(* Logix 5000 project; controller PRU vendor 1 type 14 code 107 rev 20.13; software revision 20.01; part 3 of 17 *)
(* tags used below, declared in another part *)
   LEFT_AUTO_PCNT_SETPOINT : REAL;
   Revision : DINT;
   VFD_3_Current : DINT;

ADD_ON_INSTRUCTION Totalize   (* revision 1.0, ExecuteEnableInFalse *)
// This instruction takes a flow signal (mL/min) and converts it to a total volume (mL)
VAR_INPUT
   FlowMeterCV : REAL; {required}
END_VAR
VAR_IN_OUT
   TotalVolume : REAL; {required}
END_VAR
VAR_INPUT
   FlowValve : BOOL; {required}
END_VAR
VAR_OUTPUT
   VolAddedLast : REAL; {access Read Only, visible}
END_VAR
VAR
   TOT_02 : TOTALIZER := (In := 2.289028, TimeBase := 1, Gain := 1.0, ProgProgReq := 1, ProgStopReq := 1, ProgResetReq := 1, OversampleDT := 0.5, RTSTime := 1, OldTotal := 413.70062, ProgOper := 1, ProgResetDone := 1, TargetFlag := 1, TargetDev1Flag := 1, TargetDev2Flag := 1, DeltaT := 0.001);
   BNOT_01 : FBD_BOOLEAN_NOT := (In := 1);
   __l01CE45141B44CC5A : REAL;
   __l01CE49331B44B276 : BOOL;
END_VAR

ROUTINE EnableInFalse   (* ladder *)
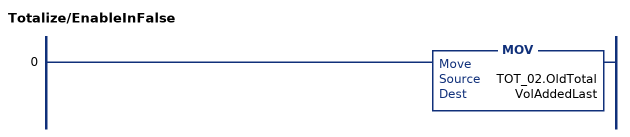
   0: MOV(TOT_02.OldTotal,VolAddedLast);
END_ROUTINE

ROUTINE Logic   (* function block diagram *)
   SHEET 1
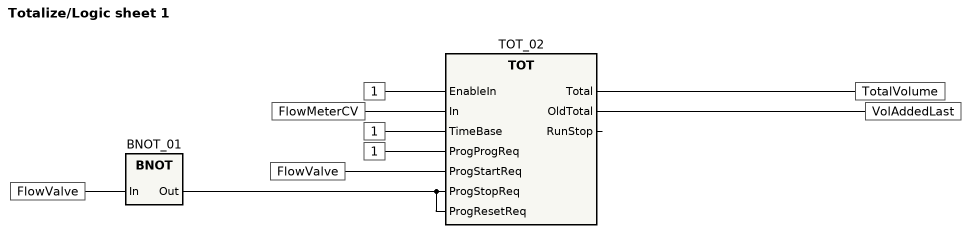
   BNOT_01 : BNOT(In := FlowValve);
   TOT_02 : TOT(EnableIn := 1, In := FlowMeterCV, TimeBase := 1, ProgProgReq := 1, ProgStartReq := FlowValve, ProgStopReq := BNOT_01.Out, ProgResetReq := BNOT_01.Out);   // unwired pins: RunStop
   TotalVolume := TOT_02.Total;
   VolAddedLast := TOT_02.OldTotal;
END_ROUTINE
END_ADD_ON_INSTRUCTION

ADD_ON_INSTRUCTION VFD_Motor_Control   (* revision 1.2, vendor Deterministic Systems, Inc. *)
// VFD Motor Control
VAR_INPUT
   IN_HARD_STOP : BOOL; {required}
   IN_HMI_STOP_PB : BOOL; {required}
   IN_RUN_INTERLOCK_1 : BOOL; {required}
   IN_RUN_INTERLOCK_2 : BOOL; {required}
   IN_RUN_INTERLOCK_3 : BOOL; {required}
   IN_VFD_IS_READY : BOOL; {required}
   IN_HMI_OFF_PB : BOOL; {required}   // Pushbutton.
   IN_HMI_MAINT_PB : BOOL; {required}   // Pushbutton.
   IN_HMI_SEMI_PB : BOOL; {required}   // Pushbutton.
   IN_HMI_AUTO_PB : BOOL; {required}   // Pushbutton.
   IN_HMI_JOG_FWD_PB : BOOL; {required}   // Pushbutton.
   IN_HMI_JOG_REV_PB : BOOL; {required}   // Pushbutton.
   IN_HMI_FWD_PB : BOOL; {required}   // Pushbutton.
   IN_HMI_REV_PB : BOOL; {required}   // Pushbutton.
   IN_HMI_AUTO_START_PB : BOOL; {required}
   IN_CURRENT_PROCESS_SEQUENCER_STEP : INT; {required}
   IN_PROCESS_SEQUENCER_AUTO_START_STEP : INT; {required}
   IN_PROCESS_SEQUENCER_AUTO_STOP_STEP : INT; {required}
   IN_HMI_SEMI_SPEED_SETPOINT_PCNT : REAL; {required}
   IN_AUTO_SPEED_SETPOINT_PERCENT : REAL; {required}
   IN_VFD_SPEED_SCALE : REAL := 6.0; {required}
   IN_VFD_ACTUAL_FREQ : REAL; {required}   // Direct from VFD.
   IN_VFD_IS_RUNNING : BOOL; {required}
END_VAR
VAR_OUTPUT
   OUT_HARD_STOPPED : BOOL; {access Read Only, required}
   OUT_OFF_MODE_ION : BOOL; {access Read Only, required}
   OUT_MAINT_MODE_ION : BOOL; {access Read Only, required}
   OUT_SEMI_MODE_ION : BOOL; {access Read Only, required}
   OUT_AUTO_MODE_ION : BOOL; {access Read Only, required}
   OUT_MODE : INT; {access Read Only, required}
   OUT_VFD_STOP_COMMAND : BOOL; {access Read Only, required}   // Direct to VFD.
   OUT_FWD_COMMAND : BOOL; {access Read Only, required}   // Direct to VFD.
   OUT_REV_COMMAND : BOOL; {access Read Only, required}   // Direct to VFD.
   OUT_JOG_COMMAND : BOOL; {access Read Only, required}   // Direct to VFD.
   OUT_VFD_RUN_COMMAND : BOOL; {access Read Only, required}   // Direct to VFD.
   OUT_CMD_RUN_ENABLED : BOOL; {access Read Only, required}   // Auto or Semi
   OUT_START_CMD_AUTO : BOOL; {access None, required}
   OUT_VFD_SPEED_SETPOINT_COMMAND : DINT; {access Read Only, required}   // Direct to VFD.
   OUT_VFD_ACTUAL_SPEED_PERCENT : REAL; {access Read Only, required}
   OUT_RUNNING_BON : BOOL; {access Read Only, required}
   OUT_RUNNING_BOF : BOOL; {access Read Only, required}
END_VAR
VAR
   AUTO_PB_ONS : BOOL; {access None}
   SEMI_PB_ONS : BOOL; {access None}
   MAINT_PB_ONS : BOOL; {access None}
   JOG_FWD_TON : TIMER := (PRE := 30000); {access None}
   LOCAL_AUTO_SETPOINT_PERCENT : REAL; {access None}
   RUNNING_TON : TIMER := (PRE := 1000); {access None}
   RUNNING_TOF : TIMER := (PRE := 1000); {access None}
END_VAR

ROUTINE Logic   (* ladder *)
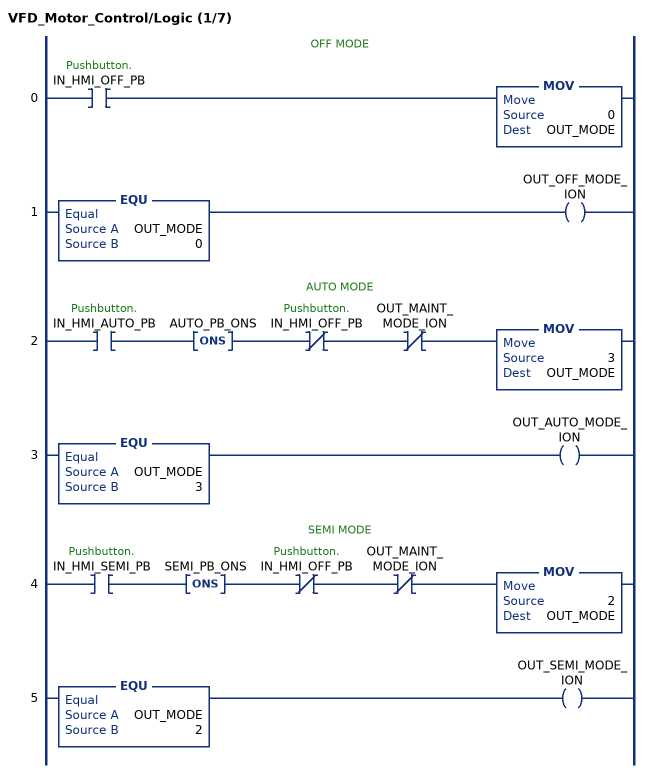
   // OFF MODE
   0: XIC(IN_HMI_OFF_PB)MOV(0,OUT_MODE);
   1: EQU(OUT_MODE,0)OTE(OUT_OFF_MODE_ION);
   // AUTO MODE
   2: XIC(IN_HMI_AUTO_PB)ONS(AUTO_PB_ONS)XIO(IN_HMI_OFF_PB)XIO(OUT_MAINT_MODE_ION)MOV(3,OUT_MODE);
   3: EQU(OUT_MODE,3)OTE(OUT_AUTO_MODE_ION);
   // SEMI MODE
   4: XIC(IN_HMI_SEMI_PB)ONS(SEMI_PB_ONS)XIO(IN_HMI_OFF_PB)XIO(OUT_MAINT_MODE_ION)MOV(2,OUT_MODE);
   5: EQU(OUT_MODE,2)OTE(OUT_SEMI_MODE_ION);
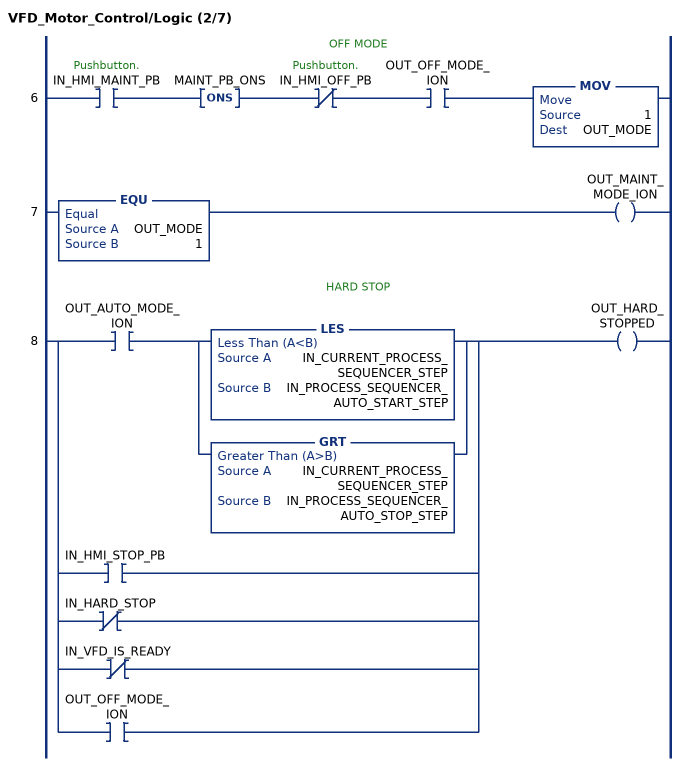
   // OFF MODE
   6: XIC(IN_HMI_MAINT_PB)ONS(MAINT_PB_ONS)XIO(IN_HMI_OFF_PB)XIC(OUT_OFF_MODE_ION)MOV(1,OUT_MODE);
   7: EQU(OUT_MODE,1)OTE(OUT_MAINT_MODE_ION);
   // HARD STOP
   8: [XIC(OUT_AUTO_MODE_ION) [LES(IN_CURRENT_PROCESS_SEQUENCER_STEP,IN_PROCESS_SEQUENCER_AUTO_START_STEP) ,GRT(IN_CURRENT_PROCESS_SEQUENCER_STEP,IN_PROCESS_SEQUENCER_AUTO_STOP_STEP) ] ,XIC(IN_HMI_STOP_PB) ,XIO(IN_HARD_STOP) ,XIO(IN_VFD_IS_READY) ,XIC(OUT_OFF_MODE_ION) ]OTE(OUT_HARD_STOPPED);
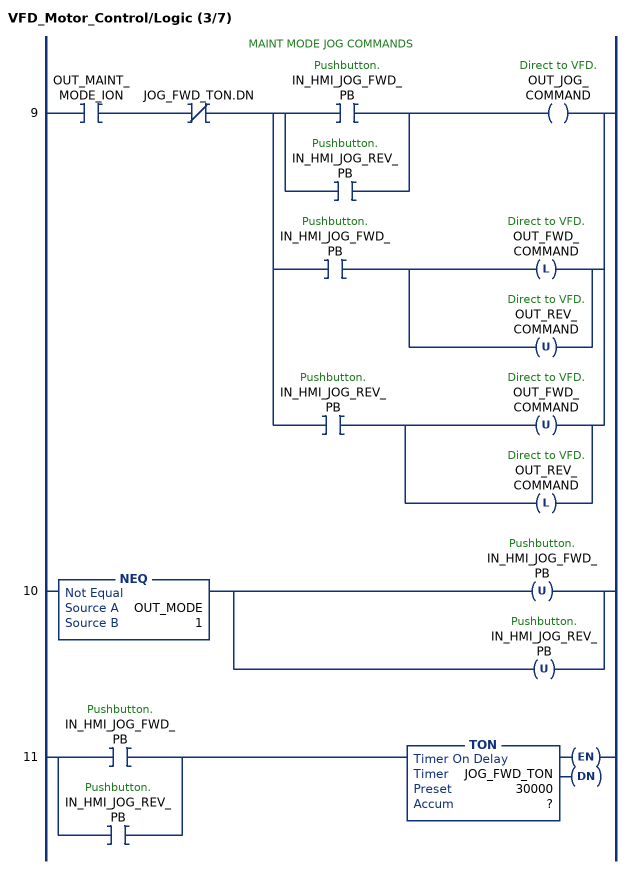
   // MAINT MODE JOG COMMANDS
   9: XIC(OUT_MAINT_MODE_ION)XIO(JOG_FWD_TON.DN)[[XIC(IN_HMI_JOG_FWD_PB) ,XIC(IN_HMI_JOG_REV_PB) ] OTE(OUT_JOG_COMMAND) ,XIC(IN_HMI_JOG_FWD_PB) [OTL(OUT_FWD_COMMAND) ,OTU(OUT_REV_COMMAND) ] ,XIC(IN_HMI_JOG_REV_PB) [OTU(OUT_FWD_COMMAND) ,OTL(OUT_REV_COMMAND) ] ];
   10: NEQ(OUT_MODE,1)[OTU(IN_HMI_JOG_FWD_PB) ,OTU(IN_HMI_JOG_REV_PB) ];
   11: [XIC(IN_HMI_JOG_FWD_PB) ,XIC(IN_HMI_JOG_REV_PB) ]TON(JOG_FWD_TON,?,?);
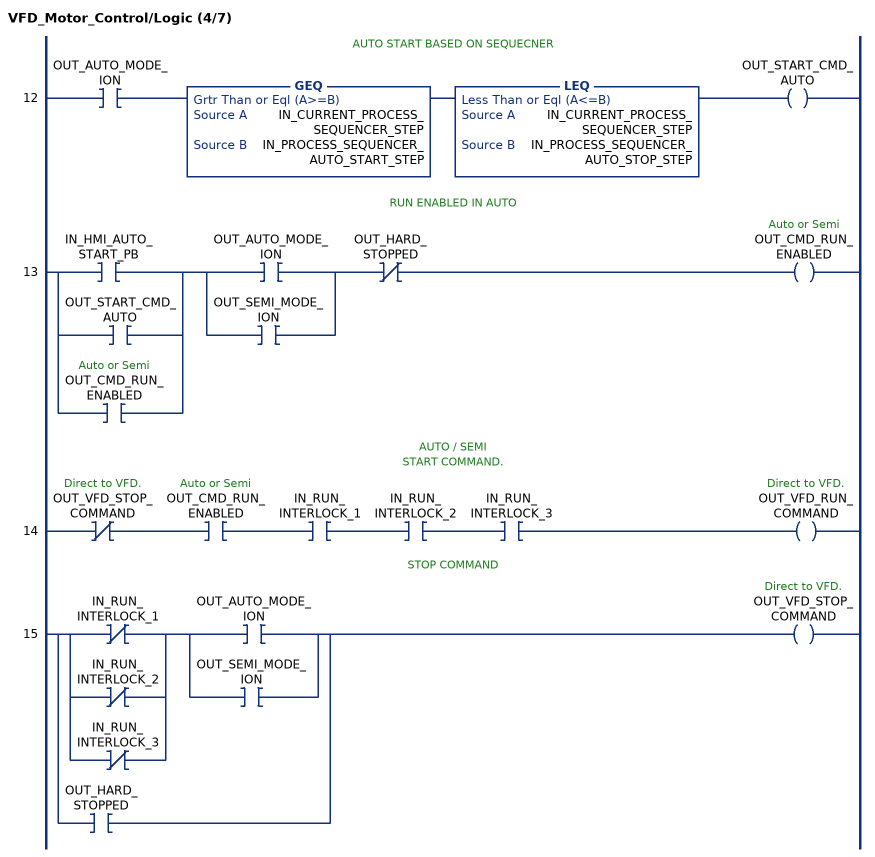
   // AUTO START BASED ON SEQUECNER
   12: XIC(OUT_AUTO_MODE_ION)GEQ(IN_CURRENT_PROCESS_SEQUENCER_STEP,IN_PROCESS_SEQUENCER_AUTO_START_STEP)LEQ(IN_CURRENT_PROCESS_SEQUENCER_STEP,IN_PROCESS_SEQUENCER_AUTO_STOP_STEP)OTE(OUT_START_CMD_AUTO);
   // RUN ENABLED IN AUTO
   13: [[XIC(IN_HMI_AUTO_START_PB) ,XIC(OUT_START_CMD_AUTO) ] ,XIC(OUT_CMD_RUN_ENABLED) ][XIC(OUT_AUTO_MODE_ION) ,XIC(OUT_SEMI_MODE_ION) ]XIO(OUT_HARD_STOPPED)OTE(OUT_CMD_RUN_ENABLED);
   // AUTO / SEMI
   // START COMMAND.
   14: XIO(OUT_VFD_STOP_COMMAND)XIC(OUT_CMD_RUN_ENABLED)XIC(IN_RUN_INTERLOCK_1)XIC(IN_RUN_INTERLOCK_2)XIC(IN_RUN_INTERLOCK_3)OTE(OUT_VFD_RUN_COMMAND);
   // STOP COMMAND
   15: [[XIO(IN_RUN_INTERLOCK_1) ,XIO(IN_RUN_INTERLOCK_2) ,XIO(IN_RUN_INTERLOCK_3) ] [XIC(OUT_AUTO_MODE_ION) ,XIC(OUT_SEMI_MODE_ION) ] ,XIC(OUT_HARD_STOPPED) ]OTE(OUT_VFD_STOP_COMMAND);
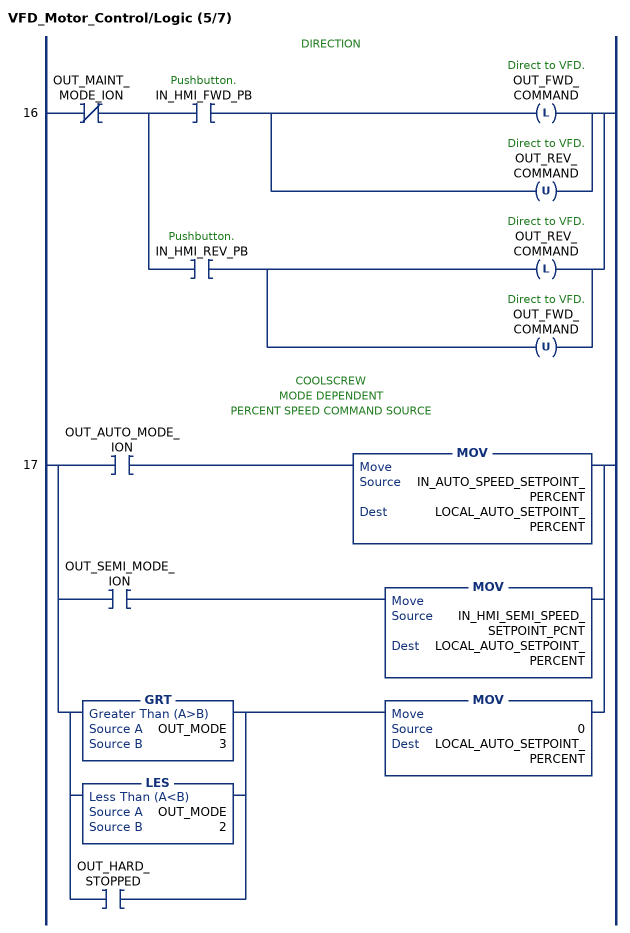
   // DIRECTION
   16: XIO(OUT_MAINT_MODE_ION)[XIC(IN_HMI_FWD_PB) [OTL(OUT_FWD_COMMAND) ,OTU(OUT_REV_COMMAND) ] ,XIC(IN_HMI_REV_PB) [OTL(OUT_REV_COMMAND) ,OTU(OUT_FWD_COMMAND) ] ];
   // COOLSCREW
   // MODE DEPENDENT
   // PERCENT SPEED COMMAND SOURCE
   17: [XIC(OUT_AUTO_MODE_ION) MOV(IN_AUTO_SPEED_SETPOINT_PERCENT,LOCAL_AUTO_SETPOINT_PERCENT) ,XIC(OUT_SEMI_MODE_ION) MOV(IN_HMI_SEMI_SPEED_SETPOINT_PCNT,LOCAL_AUTO_SETPOINT_PERCENT) ,[GRT(OUT_MODE,3) ,LES(OUT_MODE,2) ,XIC(OUT_HARD_STOPPED) ] MOV(0,LOCAL_AUTO_SETPOINT_PERCENT) ];
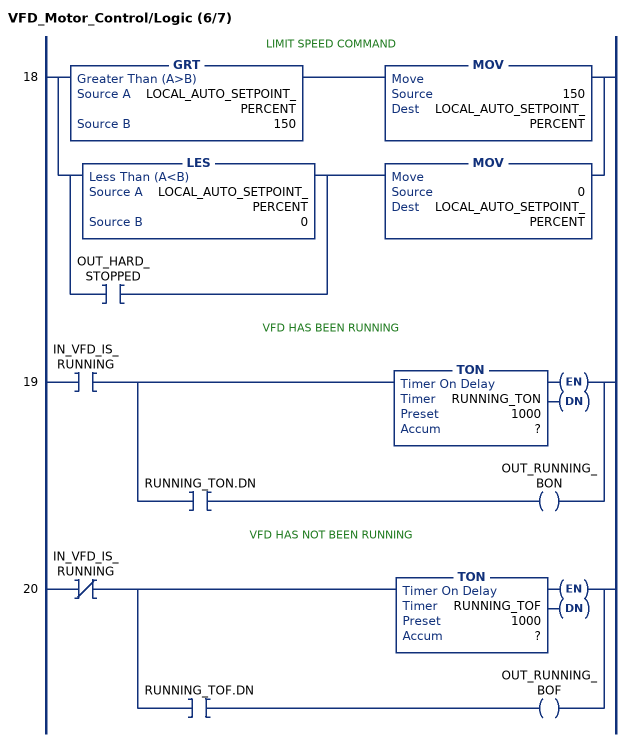
   // LIMIT SPEED COMMAND
   18: [GRT(LOCAL_AUTO_SETPOINT_PERCENT,150) MOV(150,LOCAL_AUTO_SETPOINT_PERCENT) ,[LES(LOCAL_AUTO_SETPOINT_PERCENT,0) ,XIC(OUT_HARD_STOPPED) ] MOV(0,LOCAL_AUTO_SETPOINT_PERCENT) ];
   // VFD HAS BEEN RUNNING
   19: XIC(IN_VFD_IS_RUNNING)[TON(RUNNING_TON,?,?) ,XIC(RUNNING_TON.DN) OTE(OUT_RUNNING_BON) ];
   // VFD HAS NOT BEEN RUNNING
   20: XIO(IN_VFD_IS_RUNNING)[TON(RUNNING_TOF,?,?) ,XIC(RUNNING_TOF.DN) OTE(OUT_RUNNING_BOF) ];
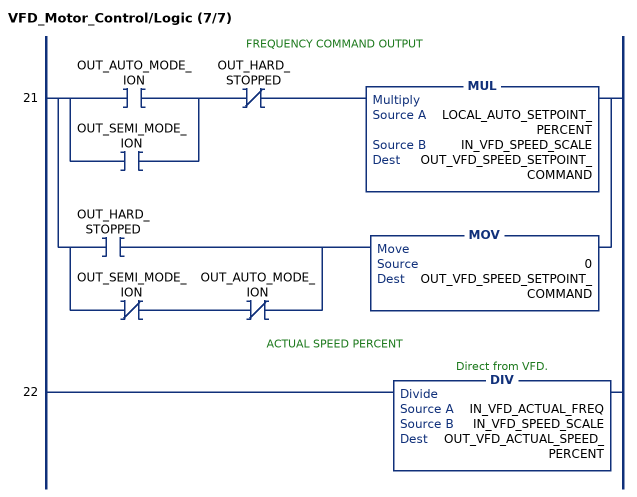
   // FREQUENCY COMMAND OUTPUT
   21: [[XIC(OUT_AUTO_MODE_ION) ,XIC(OUT_SEMI_MODE_ION) ] XIO(OUT_HARD_STOPPED) MUL(LOCAL_AUTO_SETPOINT_PERCENT,IN_VFD_SPEED_SCALE,OUT_VFD_SPEED_SETPOINT_COMMAND) ,[XIC(OUT_HARD_STOPPED) ,XIO(OUT_SEMI_MODE_ION) XIO(OUT_AUTO_MODE_ION) ] MOV(0,OUT_VFD_SPEED_SETPOINT_COMMAND) ];
   // ACTUAL SPEED PERCENT
   22: DIV(IN_VFD_ACTUAL_FREQ,IN_VFD_SPEED_SCALE,OUT_VFD_ACTUAL_SPEED_PERCENT);
END_ROUTINE
END_ADD_ON_INSTRUCTION

VAR_GLOBAL   (* controller tags *)
   ABS_ENCODER_ERROR_MINUS : REAL := 58.63318;
   ABS_ENCODER_ERROR_PLUS : REAL := 72.63318;
   ACCEL_DECEL_RAMP : REAL := 200.0;   // VFD Accel/Decel ramp rate * 10ms ie 100 * 10ms = 1sec
   ACTUAL_FWD_ION : BOOL := 1;
   ACTUAL_ILLEGAL_ION : BOOL;
   ACTUAL_REV_ION : BOOL;
   AFI : BOOL;
   Agilyx_KnifeGateIgnorePB : BOOL := 1;
   AI0_CALCULATED : REAL := 0.06;
   AI0_WF : DSi_WF50 := (IN_VALUE := 6.0, OUT_VALUE := 6.0);
   AI10_CALCULATED : REAL := 0.08;
   AI10_WF : DSi_WF50 := (IN_VALUE := 8.0, OUT_VALUE := 7.5);
   AI11_CALCULATED : REAL := 0.03;
   AI11_WF : DSi_WF50 := (OUT_VALUE := 2.88);
   AI12_CALCULATED : REAL := 0.089999996;
   AI12_WF : DSi_WF50 := (IN_VALUE := 12.0, OUT_VALUE := 9.12);
   AI13_CALCULATED : REAL := 18.56;
   AI13_WF : DSi_WF50 := (IN_VALUE := 1693.0, OUT_VALUE := 1813.78);
   AI14_CALCULATED : REAL := 19.279999;
   AI14_WF : DSi_WF50 := (IN_VALUE := 2256.0, OUT_VALUE := 2126.92);
   AI15_CALCULATED : REAL := -5.0;
   AI15_WF : DSi_WF50 := (IN_VALUE := -500.0, OUT_VALUE := -500.0);
   AI16_CALCULATED : REAL := 3.2;
   AI16_WF : DSi_WF50 := (IN_VALUE := -500.0, OUT_VALUE := -500.0);
   AI1_CALCULATED : REAL := 0.099999994;
   AI1_WF : DSi_WF50 := (IN_VALUE := 10.0, OUT_VALUE := 10.0);
   AI2_CALCULATED : REAL := 0.11;
   AI2_WF : DSi_WF50 := (IN_VALUE := 11.0, OUT_VALUE := 11.34);
   AI3_CALCULATED : REAL := 0.06;
   AI3_WF : DSi_WF50 := (IN_VALUE := 6.0, OUT_VALUE := 6.16);
   AI4_CALCULATED : REAL := 0.06;
   AI4_WF : DSi_WF50 := (IN_VALUE := 6.0, OUT_VALUE := 6.0);
   AI5_CALCULATED : REAL := 0.01;
   AI5_WF : DSi_WF50 := (IN_VALUE := 4.0, OUT_VALUE := 2.12);
   AI6_CALCULATED : REAL := 2.44;
   AI6_WF : DSi_WF50 := (IN_VALUE := 82.0, OUT_VALUE := 344.3);
   AI7_CALCULATED : REAL := 2.31;
   AI7_WF : DSi_WF50 := (IN_VALUE := 672.0, OUT_VALUE := 235.98);
   AI8_CALCULATED : REAL := 2.04;
   AI8_WF : DSi_WF50 := (IN_VALUE := 111.0, OUT_VALUE := 309.82);
   AI9_CALCULATED : REAL := 0.02;
   AI9_WF : DSi_WF50 := (IN_VALUE := -1.0, OUT_VALUE := 1.74);
   AI_0 : AI_1769_IF4 := (IN_ANALOG_INPUT_RAW := 6, IN_Ai_Hi_Scale := 100.0, IN_HMI_Ai_FORCE_VALUE := 3.0, OUT_Ai_Calc := 0.06, OUT_ANALOG_OUTPUT := 0.06);
   AI_0_FILTERED : DINT := 6;
   AI_1 : AI_1769_IF4 := (IN_ANALOG_INPUT_RAW := 10, IN_Ai_Hi_Scale := 100.0, IN_HMI_Ai_FORCE_VALUE := 3.0, OUT_Ai_Calc := 0.099999994, OUT_ANALOG_OUTPUT := 0.099999994);
   AI_10 : AI_1769_IF4 := (IN_ANALOG_INPUT_RAW := 8, IN_Ai_Hi_Scale := 100.0, OUT_Ai_Calc := 0.08, OUT_ANALOG_OUTPUT := 0.08);
   AI_10_FILTERED : REAL := 8.4;
   AI_11 : AI_1769_IF4 := (IN_ANALOG_INPUT_RAW := 2, IN_Ai_Hi_Scale := 100.0, IN_HMI_Ai_FORCE_VALUE := 33.0, OUT_Ai_Calc := 0.02, OUT_ANALOG_OUTPUT := 0.02);
   AI_11_FILTERED : REAL := 0.86;
   AI_12 : AI_1769_IF4 := (IN_ANALOG_INPUT_RAW := 9, IN_Ai_Hi_Scale := 100.0, IN_HMI_Ai_FORCE_VALUE := 42.0, OUT_Ai_Calc := 0.089999996, OUT_ANALOG_OUTPUT := 0.089999996);
   AI_12_FILTERED : REAL := 8.58;
   AI_13 : AI_1769_IF4 := (IN_ANALOG_INPUT_RAW := 1847, IN_Ai_Hi_Scale := 100.0, IN_HMI_Ai_FORCE_VALUE := 35.0, OUT_Ai_Calc := 18.47, OUT_ANALOG_OUTPUT := 18.47);
   AI_13_FILTERED : REAL := 1851.82;
   AI_14 : AI_1769_IF4 := (IN_ANALOG_INPUT_RAW := 1925, IN_Ai_Hi_Scale := 100.0, IN_HMI_Ai_FORCE_VALUE := 42.0, OUT_Ai_Calc := 19.25, OUT_ANALOG_OUTPUT := 19.25);
   AI_14_FILTERED : REAL := 1941.48;
   AI_15 : AI_1769_IF4 := (IN_ANALOG_INPUT_RAW := -500, IN_Ai_Hi_Scale := 100.0, IN_HMI_Ai_FORCE_VALUE := 37.0, OUT_Ai_Calc := -5.0, OUT_ANALOG_OUTPUT := -5.0);
   AI_15_FILTERED : REAL := -500.0;
   AI_16 : AI_1769_IF4 := (IN_ANALOG_INPUT_RAW := -500, IN_Ai_Lo_Scale := 4.0, IN_Ai_Hi_Scale := 20.0, IN_HMI_Ai_FORCE_VALUE := 50.0, OUT_Ai_Calc := 3.2, OUT_ANALOG_OUTPUT := 3.2);
   AI_16_DATA : REAL := 3.2;
   AI_16_FILTERED : REAL := -500.0;
   AI_1_FILTERED : REAL := 10.0;
   AI_2 : AI_1769_IF4 := (IN_ANALOG_INPUT_RAW := 11, IN_Ai_Hi_Scale := 100.0, IN_HMI_Ai_FORCE_VALUE := 3.0, OUT_Ai_Calc := 0.11, OUT_ANALOG_OUTPUT := 0.11);
   AI_2_FILTERED : REAL := 11.1;
   AI_3 : AI_1769_IF4 := (IN_ANALOG_INPUT_RAW := 7, IN_Ai_Hi_Scale := 100.0, IN_HMI_Ai_FORCE_VALUE := 3.0, OUT_Ai_Calc := 0.07, OUT_ANALOG_OUTPUT := 0.07);
   AI_3_FILTERED : REAL := 6.32;
   AI_4 : AI_1769_IF4 := (IN_ANALOG_INPUT_RAW := 6, IN_Ai_Hi_Scale := 100.0, IN_HMI_Ai_FORCE_VALUE := 3.0, OUT_Ai_Calc := 0.06, OUT_ANALOG_OUTPUT := 0.06);
   AI_4_FILTERED : REAL := 6.26;
   AI_5 : AI_1769_IF4 := (IN_ANALOG_INPUT_RAW := 2, IN_Ai_Hi_Scale := 100.0, IN_HMI_Ai_FORCE_VALUE := 3.0, OUT_Ai_Calc := 0.02, OUT_ANALOG_OUTPUT := 0.02);
   AI_5_FILTERED : REAL := 1.48;
   AI_6 : AI_1769_IF4 := (IN_ANALOG_INPUT_RAW := 333, IN_Ai_Hi_Scale := 100.0, IN_HMI_Ai_FORCE_VALUE := 3.0, OUT_Ai_Calc := 3.33, OUT_ANALOG_OUTPUT := 3.33);
   AI_6_FILTERED : REAL := 236.58;
   AI_7 : AI_1769_IF4 := (IN_ANALOG_INPUT_RAW := 224, IN_Ai_Hi_Scale := 100.0, IN_HMI_Ai_FORCE_VALUE := 3.0, OUT_Ai_Calc := 2.24, OUT_ANALOG_OUTPUT := 2.24);
   AI_7_FILTERED : REAL := 233.06;
   AI_8 : AI_1769_IF4 := (IN_ANALOG_INPUT_RAW := 275, IN_Ai_Hi_Scale := 100.0, IN_HMI_Ai_FORCE_VALUE := 10.0, OUT_Ai_Calc := 2.75, OUT_ANALOG_OUTPUT := 2.75);
   AI_8_FILTERED : REAL := 198.48;
   AI_9 : AI_1769_IF4 := (IN_ANALOG_INPUT_RAW := 2, IN_Ai_Hi_Scale := 100.0, IN_HMI_Ai_FORCE_VALUE := 15.0, OUT_Ai_Calc := 0.02, OUT_ANALOG_OUTPUT := 0.02);
   AI_9_FILTERED : REAL := 1.4;
   AlarmMaster : DINT;
        .0   // MESSAGE ALARM bit.0
        .1   // WARNING ALARM bit.1
        .2   // CSS_START_DISABLE bit.2
        .3   // PRU_START_DISABLE bit.3
        .4   // PRU_RUN_DISABLE bit.4
   AlarmMasterDisable : BOOL;
   AlarmMasterResetTON : TIMER := (PRE := 1000, ACC := 689, EN := 1, TT := 1);
   AlarmResetPB : BOOL;
   ALL_AUTO_IOK : BOOL := 1;   // All equipment is in Auto Mode.
   ALL_DRIVES_ARE_CMD_FWD : BOOL := 1;
   ALL_DRIVES_ARE_READY : BOOL := 1;
   ALL_SHUTDOWN_FAULTS_IOK : BOOL := 1;
   AUTO_DISCHARGE_CYCLE_ION : BOOL := 1;   // Proces Sequencer (4-13)
   AUTO_FWD_CMD : BOOL;
   AUTO_FWD_CMD_GON : BOOL := 1;
   AUTO_FWD_CMD_GON_VALUE : DINT := 3;
   AUTO_FWD_CMD_VALUE : DINT;
   AUTO_SHUTDOWN_ENABLE : BOOL := 1;
   CALC_SPARE_AO_CMD : REAL := 50.0;
   CENTERING_BON : BOOL;
   CENTERING_BON_ONS : BOOL;
   CENTERING_BON_SS : BOOL;
   CENTERING_ERROR : REAL;
   CENTERING_ERROR_NOW : REAL;
   CENTERING_ERROR_WAS : REAL;
   CENTERING_ONS : BOOL;
   CENTERING_SS : BOOL;
   CENTERING_TON : TIMER := (PRE := 1000);
   CHANGING_TOTE : BOOL;
   CHANGING_TOTE_1 : BOOL;
   CHANGING_TOTE_2 : BOOL;
   CHANGING_TOTE_3 : BOOL;
   CHANGING_TOTE_4 : BOOL;
   CHANGING_TOTE_5 : BOOL;
   CLEARING_PYROLIZER_TIME_REMAINING_SEC : REAL := 60.0;
   CLEARING_PYROLIZER_TIME_REMAINING_TEMP : REAL := 60000.0;
   CLEARING_PYROLIZER_TIMER : TIMER := (PRE := 60000);
   CMD_LEFT_SCREW_START : BOOL;
   CMD_LEFT_SCREW_STOP : BOOL;
   CMD_RIGHT_SCREW_START : BOOL;
   CMD_RIGHT_SCREW_STOP : BOOL;
   CONTROLLED_STOP : BOOL;
   COOL_FOR_MOTOR_STOP : BOOL;
   COOL_MESSAGE_FON1 : TIMER := (PRE := 1000);
   COOL_MESSAGE_FON2 : TIMER := (PRE := 1000, ACC := 248, EN := 1, TT := 1);
   COOL_VFD_Message : MESSAGE;
        MessageParameters(ServiceCode := 16#000e, DestinationTag := VFD_3_Current, ...)
   COOLSCREW : VFD := (MODE := 3, SPEED_SETPOINT_SEMI := 40.0, SPEED_SETPOINT_AUTO := 40.0, INTERLOCK_1 := 1, INTERLOCK_2 := 1, INTERLOCK_3 := 1, ACTUAL_SPEED := 40.0, ACTUAL_SPEED_CONVERSION_FACTOR := 6.0, MODE_AUTO_ION := 1, VFD_BEEN_ON := 1, CMD_AUTO_RUN_ENABLED := 1, CMD_AUTO_STARTED := 1);
   CR0_CON1_HTR1_GON : BOOL := 1;   // ZONE 1 (L1,L2,L3)
   CR0_CON1_HTR1_LON : BOOL := 1;   // AUTO LOGIC - ZONE 1 HEATER CONTACTOR
   CR1_CON2_HTR2_GON : BOOL := 1;   // ZONE 2 (L1,L2,L3)
   CR1_CON2_HTR2_LON : BOOL := 1;   // AUTO LOGIC - ZONE 2 HEATER CONTACTOR
   CR2_CON3_HTR3_GON : BOOL := 1;   // ZONE 3 (L1,L2,L3)
   CR2_CON3_HTR3_LON : BOOL := 1;   // AUTO LOGIC - ZONE 3 HEATER CONTACTOR
   CR3_CON4_HTR4_GON : BOOL := 1;   // ZONE 4 (L1) ZONE 5 (L2) ZONE 6 (L3)
   CR3_CON4_HTR4_LON : BOOL := 1;   // AUTO LOGIC - ZONES 4-6 HEATER CONTACTOR
   CR4_CON5_HTR5_GON : BOOL := 1;   // ZONE 7 (L1) ZONE 8 (L2) ZONE 9 (L3)
   CR4_CON5_HTR5_LON : BOOL := 1;   // AUTO LOGIC - ZONES 7-9 HEATER CONTACTOR
   CR5_CON1_SAFETY_GON : BOOL := 1;
   CR5_CON1_SAFETY_LON : BOOL := 1;
   CR6_CON2_SAFETY_GON : BOOL := 1;
   CR6_CON2_SAFETY_LON : BOOL := 1;
   CR7_VFD_DRYERL_GON : BOOL := 1;
   CR7_VFD_DRYERL_LON : BOOL := 1;
   CR8_VFD_DRYERR_GON : BOOL;
   CR8_VFD_DRYERR_LON : BOOL;
   CSS_CommsLoss_TMR : TIMER := (PRE := 60000, EN := 1, TT := 1);
   CSS_CommsLossAlm : BOOL;
   CSS_CommsWarning_TMR : TIMER := (PRE := 5000);
   CSS_CommsWarningAlm : BOOL;
   CSS_PLC_Seconds_Temp : DINT := 6;
   CSS_Status_Data : PLCStatusData := (PLCSenonds := 12, AlarmMaster := 2, Status[0] := 403, Status[1] := 723, Status[2] := 623, Status[3] := -1872, Status[4] := -1995, Status[5] := -2109, Status[6] := 8414, Status[7] := -4146, Status[8] := -4000);
   CYCLE_ION_DELAY1_TON : TIMER := (PRE := 2000, ACC := 2001, EN := 1, DN := 1);
   CYCLE_ION_DELAY2_TON : TIMER := (PRE := 2000, ACC := 2006, EN := 1, DN := 1);
   CYCLE_ION_DELAY3_TON : TIMER := (PRE := 2000, ACC := 2000, EN := 1, DN := 1);
   CYCLE_ION_DELAY4_TON : TIMER := (PRE := 2000, ACC := 2003, EN := 1, DN := 1);
   CYCLE_START_ONS : BOOL;
   CYCLE_START_SS : BOOL;   // Begin temperature ramp and hold heat cycle.
   DailyTotalResetPB : BOOL := 1;
   DATA_RECORD_INDEX : INT;
   DCS_ESTOP_ION : BOOL := 1;
   DI0_ION : BOOL := 1;
   DI10_ION : BOOL;
   DI11_ION : BOOL := 1;
   DI12_ION : BOOL;
   DI13_ION : BOOL := 1;
   DI14_ION : BOOL;
   DI15_ION : BOOL := 1;
   DI16_ION : BOOL;
   DI17_ION : BOOL;
   DI18_ION : BOOL := 1;
   DI19_ION : BOOL := 1;
   DI1_ION : BOOL := 1;
   DI20_ION : BOOL := 1;
   DI21_ION : BOOL;
   DI22_ION : BOOL := 1;
   DI23_ION : BOOL;
   DI24_ION : BOOL;
   DI25_ION : BOOL;
   DI26_ION : BOOL;
   DI27_ION : BOOL := 1;
   DI28_ION : BOOL;
   DI29_ION : BOOL;
   DI2_ION : BOOL := 1;
   DI30_ION : BOOL;
   DI31_ION : BOOL;
   DI3_ION : BOOL := 1;
   DI4_ION : BOOL := 1;
   DI5_ION : BOOL := 1;
   DI6_ION : BOOL := 1;
   DI7_ION : BOOL;
   DI8_ION : BOOL;
   DI9_ION : BOOL;
   DisableAllHeaters : BOOL;
   DRYER : DUAL_SCREW := (HMI_AUTO_SCREW_CMD_PCNT := 34.0, AUTO_SCREW_RIGHT_CMD_PCNT := 33.2266, LEFT_ENCODER_G := 3567, RIGHT_ENCODER_G := 559, LEFT_ENCODER_DEG_IS := 209.0039, RIGHT_ENCODER_DEG_IS := 274.7461, LEFT_AUTO_PCNT_SETPOINT := 34.0);
   DRYER_AUTO_MODE_PB_ONS : BOOL;
   DRYER_CENTER_STARTUP_MODE : BOOL;
   DRYER_CENTER_TON : TIMER := (PRE := 2000);
   DRYER_FWD_MODE : BOOL := 1;
   DRYER_IS_CENTERING : BOOL;
   DRYER_MAN_MODE_PB_ONS : BOOL;
   DRYER_MODE_AUTO : BOOL := 1;
   DRYER_MODE_OFF : BOOL;
   DRYER_ONS : BOOL := 1;
   DRYER_SEMIAUTO_MODE_PB_ONS : BOOL;
   DRYER_SHUTDOWN_FAULT_ION : BOOL;
   DRYERL_ACTUAL_SPEED : REAL := 16.0037;
   DRYERR_ACTUAL_SPEED : REAL := 12.937757;
   DUMMY_REAL : REAL;
   ENCODER_ACC : REAL := 14.501953;
   ENCODER_ERROR : REAL := 65.63008;
   ENCODER_OFFSET : REAL := -0.2;
   ENCODER_RATE : REAL := 14.501953;
   ESR_CONTACT_1_ION : BOOL := 1;
   ESR_CONTACT_2_ION : BOOL := 1;
   ESR_CONTACT_3_ION : BOOL;
   ESR_RESET_PB_ION : BOOL;
   ESTOP_PB_IOF : BOOL;   // E-STOP PUSHBUTTON IS PUSHED.
   FAULT : DINT[100];
        [9].0   // Changing Char Tote 1 Longer than 30 min
   FAULT_31_14_ONS : BOOL;
   FAULT_DRYERL_MSG_TON : TIMER := (PRE := 1000, ACC := 20, EN := 1, TT := 1);
   FAULT_DRYERR_MSG_TON : TIMER := (PRE := 1000, ACC := 20, EN := 1, TT := 1);
   FAULT_TIMER : TIMER[10000] := ([108].PRE := 5000, [109].PRE := 5000, [110].PRE := 5000, [111].PRE := 5000, [112].PRE := 5000, [113].PRE := 5000, [114].PRE := 5000, [115].PRE := 5000, [116].PRE := 5000, [117].PRE := 5000, [118].PRE := 5000, [119].PRE := 5000, [404].PRE := 5000, [500].PRE := 3000, [501].PRE := 3000, [600].PRE := 2000, [601].PRE := 2000, [602].PRE := 2000, [603].PRE := 2000, [604].PRE := 2000, [605].PRE := 2000, [606].PRE := 2000, [607].PRE := 2000, [608].PRE := 2000, [609].PRE := 2000, [610].PRE := 2000, [611].PRE := 2000, [612].PRE := 2000, [613].PRE := 2000, [614].PRE := 2000, [615].PRE := 2000, [616].PRE := 2000, [617].PRE := 2000, [618].PRE := 2000, [619].PRE := 2000, [620].PRE := 2000, [621].PRE := 2000, [622].PRE := 2000, [623].PRE := 2000, [624].PRE := 2000, [625].PRE := 2000, [626].PRE := 2000, [627].PRE := 2000, [628].PRE := 2000, [629].PRE := 2000, [630].PRE := 2000, [631].PRE := 2000, [700].PRE := 2000, [701].PRE := 2000, [702].PRE := 2000, [703].PRE := 2000, [704].PRE := 2000, [705].PRE := 2000, [706].PRE := 2000, [707].PRE := 2000, [708].PRE := 2000, [709].PRE := 2000, [710].PRE := 2000, [711].PRE := 2000, [712].PRE := 2000,
        [713].PRE := 2000, [714].PRE := 2000, [715].PRE := 2000, [716].PRE := 2000, [717].PRE := 2000, [718].PRE := 2000, [719].PRE := 2000, [720].PRE := 2000, [721].PRE := 2000, [722].PRE := 2000, [723].PRE := 2000, [724].PRE := 2000, [725].PRE := 2000, [726].PRE := 2000, [727].PRE := 2000, [728].PRE := 2000, [729].PRE := 2000, [730].PRE := 2000, [731].PRE := 2000, [800].PRE := 10000, [801].PRE := 10000, [3001].PRE := 1000, [3001].ACC := 10, [3001].EN := 1, [3001].TT := 1, [3002].PRE := 1000, [3004].PRE := 1500, [3006].PRE := 1500, [3007].PRE := 1500, [3010].PRE := 12000, [3011].PRE := 20, [3012].PRE := 20, [3014].PRE := 3000, [3016].PRE := 1000, [3017].PRE := 3000, [3019].PRE := 1500, [3020].PRE := 12000, [3021].PRE := 1500, [3022].PRE := 3000, [3025].PRE := 12000, [3026].PRE := 20, [3027].PRE := 20, [3029].PRE := 20, [3030].PRE := 2000, [3031].PRE := 1000, [3102].PRE := 1000, [3103].PRE := 1000, [3108].PRE := 5000, [3109].PRE := 5000, [3112].PRE := 100, [3113].PRE := 100, [3114].PRE := 1000, [4000].PRE := 2000, [4001].PRE := 2000, [4002].PRE := 2000, [4003].PRE := 2000, [4004].PRE := 2000, [4005].PRE := 2000, [4006].PRE := 2000, [4007].PRE := 2000,
        [4008].PRE := 2000, [4009].PRE := 2000, [4010].PRE := 2000, [4011].PRE := 2000, [4012].PRE := 2000, [4013].PRE := 2000, [4014].PRE := 2000, [4015].PRE := 2000, [4016].PRE := 2000, [4017].PRE := 2000, [4018].PRE := 2000, [4019].PRE := 2000, [4020].PRE := 2000, [4021].PRE := 2000, [4022].PRE := 2000, [4023].PRE := 2000, [4024].PRE := 2000, [4025].PRE := 2000, [4026].PRE := 2000, [4027].PRE := 2000, [4028].PRE := 2000, [4029].PRE := 2000, [4030].PRE := 2000, [4031].PRE := 2000, [5004].PRE := 2000, [5005].PRE := 20000, [5006].PRE := 3000, [5007].PRE := 3000, [5008].PRE := 2000, [5009].PRE := 10000, [5010].ACC := 4, [5010].EN := 1, [5010].DN := 1, [5800].PRE := 3000, [5801].PRE := 3000, [5802].PRE := 3000, [5803].PRE := 3000, [5804].PRE := 3000, [5805].PRE := 2000, [5806].PRE := 2000, [5807].PRE := 2000, [5808].PRE := 2000, [5809].PRE := 2000, [5810].PRE := 2000, [5811].PRE := 2000, [5812].PRE := 2000, [5813].PRE := 2000, [5814].PRE := 2000, [5815].PRE := 2000, [5816].PRE := 2000, [5817].PRE := 2000, [5818].PRE := 2000, [5819].PRE := 2000, [6500].PRE := 2000, [6501].PRE := 30000, [6502].PRE := 30000, [6503].PRE := 2000, [6600].PRE := 2000, [6601].PRE := 30000, [6602].PRE := 30000,
        [6603].PRE := 2000);
   FAULT_TIMER_3112_TmrExtended : BOOL;
   FAULT_TIMER_3112_TmrNormal : BOOL := 1;
   FAULTS_FA1_IOK : BOOL := 1;   // SYSTEM LEVEL FAULTS ARE OK.
   FAULTS_FA1A_IOK : BOOL := 1;   // MODULE FAULTS ARE OK.
   FAULTS_FA1B_IOK : BOOL := 1;   // STOP PUSHBUTTON FAULTS ARE OK.
   FAULTS_FA3_IOK : BOOL := 1;
   FAULTS_FA3A_IOK : BOOL := 1;   // SCREWS DRIVES NOT FAULTED.
   FAULTS_FA3B_IOK : BOOL := 1;   // ENCODERS NOT FAULTED.
   FAULTS_FA4_IOK : BOOL := 1;   // HI TEMP FAULTS ARE OK.
   FAULTS_FA4A_IOK : BOOL := 1;   // HIGH TEMPERATURE FAULTS ARE OK.
   FAULTS_FA5_IOK : BOOL := 1;
   FAULTS_FA5A_IOK : BOOL := 1;   // COOLING SCREW FAULTS ARE OK.
   FAULTS_FA5C_IOK : BOOL := 1;   // KG021 FAULTS ARE OK.
   FAULTS_FA5D_IOK : BOOL := 1;   // KG021 FAULTS ARE OK.
   FAULTS_FA6_IOK : BOOL := 1;   // HEATER FAULTS ARE OK.
   FAULTS_FA6A_IOK : BOOL := 1;
   FAULTS_FA6B_IOK : BOOL := 1;
   FEED_DWELL_DEG : INT;
   FEED_IS_DWELLING : BOOL := 1;
   FEED_SHOT_ENABLE_Enabled : BOOL := 1;
   FEED_SHOT_ENABLE_GON : BOOL;
   FEED_SHOT_ENABLE_GON_ONS : BOOL := 1;
   FEED_SHOT_ENABLE_GON_Tmr : TIMER := (PRE := 9999999, ACC := 12989);
   FEED_SHOT_ENABLE_GON_TmrONS : BOOL;
   FEED_SHOT_ENABLE_GON_TmrONS1 : BOOL;
   FEED_SHOT_ENABLE_GON_TmrONS2 : BOOL := 1;
   FEED_SHOT_ENABLE_ONS : BOOL := 1;
   FEED_SHOT_ENABLE_ONSN : BOOL;
   FEED_SHOT_ENABLE_SS : BOOL;
   FEED_SHOT_ENABLE_SSN : BOOL;
   FEED_TIME : REAL := 45.0;
   FEED_TIME_OFF : TIMER := (PRE := 45000);
   FEED_TIME_OFF_DSEC : REAL := 4000.0;
   FEED_TIME_OFF_REM : REAL := 45.0;
   FEED_TIME_OFF_REM_TEMP : REAL := 45000.0;
   FEED_TIME_OFF_SEC : REAL := 45.0;
   FEED_TIME_ON : TIMER;
   FEED_TIME_ON_REM : REAL;
   FEED_TIME_ON_REM_TEMP : REAL;
   FEED_TIME_ON_SEC : REAL;
   FEED_TRIGGER : BOOL := 1;
   FEED_UNWIND_THRESHOLD : INT := 145;
   FINISH_PROCESS_TIME_REMAINING_SEC : REAL := 120.0;
   FINISH_PROCESS_TIME_REMAINING_TEMP : REAL := 120000.0;
   FINISH_PROCESS_TIMER : TIMER := (PRE := 120000);
   FIRST_CYCLE : BOOL;
   FS0101_ION : BOOL := 1;   // LOW FLOW SWITCH - INLET AND DISCHARGE PURGE
   FS0102H_ION : BOOL := 1;   // HIGH FLOW SWITCH - DISCHARGE END SHAFT SEAL
   FS0102L_ION : BOOL := 1;   // LOW FLOW SWITCH - DISCHARGE END SHAFT SEAL
   FS0103H_ION : BOOL := 1;   // HIGH FLOW SWITCH - CHAMBER END INLET SEALS
   FS0103L_ION : BOOL := 1;   // LOW FLOW SWITCH - CHAMBER END INLET SEALS
   FS0201_ION : BOOL;   // LOW FLOW SWITCH - KG021 PURGE
   FS0202_ION : BOOL := 1;   // LOW FLOW SWITCH - KG022 PURGE
   FS0203H_ION : BOOL := 1;   // HIGH FLOW SWITCH - COOLING SHAFT SEALS
   FS0203L_ION : BOOL := 1;   // LOW FLOW SWITCH - COOLING SHAFT SEALS
   FS0204_ION : BOOL := 1;   // LOW FLOW SWITCH - COOLING SCREW COOLING WATER
   FWD_CMD_BON : TIMER := (PRE := 1500, ACC := 1506, EN := 1, DN := 1);
   FWD_SCAN_COUNT : DINT := 12989;
   FWD_SCAN_COUNTING : DINT := 2532;
   FWD_SCAN_SEC : REAL := 12.989;
   GRAY : REAL[4097] := ([1] := 0.087890625, [2] := 0.26367188, [3] := 0.17578125, [4] := 0.6152344, [5] := 0.52734375, [6] := 0.3515625, [7] := 0.43945312, [8] := 1.3183594, [9] := 1.2304688, [10] := 1.0546875, [11] := 1.1425781, [12] := 0.703125, [13] := 0.7910156, [14] := 0.9667969, [15] := 0.87890625, [16] := 2.7246094, [17] := 2.6367188, [18] := 2.4609375, [19] := 2.5488281, [20] := 2.109375, [21] := 2.1972656, [22] := 2.3730469, [23] := 2.2851562, [24] := 1.40625, [25] := 1.4941406, [26] := 1.6699219, [27] := 1.5820312, [28] := 2.0214844, [29] := 1.9335938, [30] := 1.7578125, [31] := 1.8457031, [32] := 5.5371094, [33] := 5.4492188, [34] := 5.2734375, [35] := 5.361328, [36] := 4.921875, [37] := 5.0097656, [38] := 5.185547, [39] := 5.0976562, [40] := 4.21875, [41] := 4.3066406, [42] := 4.482422, [43] := 4.3945312, [44] := 4.8339844, [45] := 4.7460938, [46] := 4.5703125, [47] := 4.658203, [48] := 2.8125, [49] := 2.9003906, [50] := 3.0761719, [51] := 2.9882812, [52] := 3.4277344, [53] := 3.3398438, [54] := 3.1640625, [55] := 3.2519531, [56] := 4.1308594, [57] := 4.0429688, [58] := 3.8671875, [59] := 3.9550781, [60] := 3.515625,
        [61] := 3.6035156, [62] := 3.7792969, [63] := 3.6914062, [64] := 11.162109, [65] := 11.074219, [66] := 10.8984375, [67] := 10.986328, [68] := 10.546875, [69] := 10.634766, [70] := 10.810547, [71] := 10.722656, [72] := 9.84375, [73] := 9.931641, [74] := 10.107422, [75] := 10.019531, [76] := 10.458984, [77] := 10.371094, [78] := 10.1953125, [79] := 10.283203, [80] := 8.4375, [81] := 8.525391, [82] := 8.701172, [83] := 8.613281, [84] := 9.052734, [85] := 8.964844, [86] := 8.7890625, [87] := 8.876953, [88] := 9.755859, [89] := 9.667969, [90] := 9.4921875, [91] := 9.580078, [92] := 9.140625, [93] := 9.228516, [94] := 9.404297, [95] := 9.316406, [96] := 5.625, [97] := 5.7128906, [98] := 5.888672, [99] := 5.8007812, [100] := 6.2402344, [101] := 6.1523438, [102] := 5.9765625, [103] := 6.064453, [104] := 6.9433594, [105] := 6.8554688, [106] := 6.6796875, [107] := 6.767578, [108] := 6.328125, [109] := 6.4160156, [110] := 6.591797, [111] := 6.5039062, [112] := 8.349609, [113] := 8.261719, [114] := 8.0859375, [115] := 8.173828, [116] := 7.734375, [117] := 7.8222656, [118] := 7.998047, [119] := 7.9101562, [120] := 7.03125,
        [121] := 7.1191406, [122] := 7.294922, [123] := 7.2070312, [124] := 7.6464844, [125] := 7.5585938, [126] := 7.3828125, [127] := 7.470703, [128] := 22.41211, [129] := 22.324219, [130] := 22.148438, [131] := 22.236328, [132] := 21.796875, [133] := 21.884766, [134] := 22.060547, [135] := 21.972656, [136] := 21.09375, [137] := 21.18164, [138] := 21.357422, [139] := 21.269531, [140] := 21.708984, [141] := 21.621094, [142] := 21.445312, [143] := 21.533203, [144] := 19.6875, [145] := 19.77539, [146] := 19.951172, [147] := 19.863281, [148] := 20.302734, [149] := 20.214844, [150] := 20.039062, [151] := 20.126953, [152] := 21.00586, [153] := 20.917969, [154] := 20.742188, [155] := 20.830078, [156] := 20.390625, [157] := 20.478516, [158] := 20.654297, [159] := 20.566406, [160] := 16.875, [161] := 16.96289, [162] := 17.138672, [163] := 17.050781, [164] := 17.490234, [165] := 17.402344, [166] := 17.226562, [167] := 17.314453, [168] := 18.19336, [169] := 18.105469, [170] := 17.929688, [171] := 18.017578, [172] := 17.578125, [173] := 17.666016, [174] := 17.841797, [175] := 17.753906, [176] := 19.59961, [177] := 19.511719, [178] := 19.335938, [179] := 19.423828, [180] := 18.984375,
        [181] := 19.072266, [182] := 19.248047, [183] := 19.160156, [184] := 18.28125, [185] := 18.36914, [186] := 18.544922, [187] := 18.457031, [188] := 18.896484, [189] := 18.808594, [190] := 18.632812, [191] := 18.720703, [192] := 11.25, [193] := 11.337891, [194] := 11.513672, [195] := 11.425781, [196] := 11.865234, [197] := 11.777344, [198] := 11.6015625, [199] := 11.689453, [200] := 12.568359, [201] := 12.480469, [202] := 12.3046875, [203] := 12.392578, [204] := 11.953125, [205] := 12.041016, [206] := 12.216797, [207] := 12.128906, [208] := 13.974609, [209] := 13.886719, [210] := 13.7109375, [211] := 13.798828, [212] := 13.359375, [213] := 13.447266, [214] := 13.623047, [215] := 13.535156, [216] := 12.65625, [217] := 12.744141, [218] := 12.919922, [219] := 12.832031, [220] := 13.271484, [221] := 13.183594, [222] := 13.0078125, [223] := 13.095703, [224] := 16.78711, [225] := 16.699219, [226] := 16.523438, [227] := 16.611328, [228] := 16.171875, [229] := 16.259766, [230] := 16.435547, [231] := 16.347656, [232] := 15.46875, [233] := 15.556641, [234] := 15.732422, [235] := 15.644531, [236] := 16.083984, [237] := 15.996094, [238] := 15.8203125, [239] := 15.908203, [240] := 14.0625,
        [241] := 14.150391, [242] := 14.326172, [243] := 14.238281, [244] := 14.677734, [245] := 14.589844, [246] := 14.4140625, [247] := 14.501953, [248] := 15.380859, [249] := 15.292969, [250] := 15.1171875, [251] := 15.205078, [252] := 14.765625, [253] := 14.853516, [254] := 15.029297, [255] := 14.941406, [256] := 44.91211, [257] := 44.82422, [258] := 44.648438, [259] := 44.73633, [260] := 44.296875, [261] := 44.384766, [262] := 44.560547, [263] := 44.472656, [264] := 43.59375, [265] := 43.68164, [266] := 43.85742, [267] := 43.76953, [268] := 44.208984, [269] := 44.121094, [270] := 43.945312, [271] := 44.033203, [272] := 42.1875, [273] := 42.27539, [274] := 42.45117, [275] := 42.36328, [276] := 42.802734, [277] := 42.714844, [278] := 42.539062, [279] := 42.626953, [280] := 43.50586, [281] := 43.41797, [282] := 43.242188, [283] := 43.33008, [284] := 42.890625, [285] := 42.978516, [286] := 43.154297, [287] := 43.066406, [288] := 39.375, [289] := 39.46289, [290] := 39.63867, [291] := 39.55078, [292] := 39.990234, [293] := 39.902344, [294] := 39.726562, [295] := 39.814453, [296] := 40.69336, [297] := 40.60547, [298] := 40.429688, [299] := 40.51758, [300] := 40.078125,
        [301] := 40.166016, [302] := 40.341797, [303] := 40.253906, [304] := 42.09961, [305] := 42.01172, [306] := 41.835938, [307] := 41.92383, [308] := 41.484375, [309] := 41.572266, [310] := 41.748047, [311] := 41.660156, [312] := 40.78125, [313] := 40.86914, [314] := 41.04492, [315] := 40.95703, [316] := 41.396484, [317] := 41.308594, [318] := 41.132812, [319] := 41.220703, [320] := 33.75, [321] := 33.83789, [322] := 34.01367, [323] := 33.92578, [324] := 34.365234, [325] := 34.277344, [326] := 34.101562, [327] := 34.189453, [328] := 35.06836, [329] := 34.98047, [330] := 34.804688, [331] := 34.89258, [332] := 34.453125, [333] := 34.541016, [334] := 34.716797, [335] := 34.628906, [336] := 36.47461, [337] := 36.38672, [338] := 36.210938, [339] := 36.29883, [340] := 35.859375, [341] := 35.947266, [342] := 36.123047, [343] := 36.035156, [344] := 35.15625, [345] := 35.24414, [346] := 35.41992, [347] := 35.33203, [348] := 35.771484, [349] := 35.683594, [350] := 35.507812, [351] := 35.595703, [352] := 39.28711, [353] := 39.19922, [354] := 39.023438, [355] := 39.11133, [356] := 38.671875, [357] := 38.759766, [358] := 38.935547, [359] := 38.847656, [360] := 37.96875,
        [361] := 38.05664, [362] := 38.23242, [363] := 38.14453, [364] := 38.583984, [365] := 38.496094, [366] := 38.320312, [367] := 38.408203, [368] := 36.5625, [369] := 36.65039, [370] := 36.82617, [371] := 36.73828, [372] := 37.177734, [373] := 37.089844, [374] := 36.914062, [375] := 37.001953, [376] := 37.88086, [377] := 37.79297, [378] := 37.617188, [379] := 37.70508, [380] := 37.265625, [381] := 37.353516, [382] := 37.529297, [383] := 37.441406, [384] := 22.5, [385] := 22.58789, [386] := 22.763672, [387] := 22.675781, [388] := 23.115234, [389] := 23.027344, [390] := 22.851562, [391] := 22.939453, [392] := 23.81836, [393] := 23.730469, [394] := 23.554688, [395] := 23.642578, [396] := 23.203125, [397] := 23.291016, [398] := 23.466797, [399] := 23.378906, [400] := 25.22461, [401] := 25.136719, [402] := 24.960938, [403] := 25.048828, [404] := 24.609375, [405] := 24.697266, [406] := 24.873047, [407] := 24.785156, [408] := 23.90625, [409] := 23.99414, [410] := 24.169922, [411] := 24.082031, [412] := 24.521484, [413] := 24.433594, [414] := 24.257812, [415] := 24.345703, [416] := 28.03711, [417] := 27.949219, [418] := 27.773438, [419] := 27.861328, [420] := 27.421875,
        [421] := 27.509766, [422] := 27.685547, [423] := 27.597656, [424] := 26.71875, [425] := 26.80664, [426] := 26.982422, [427] := 26.894531, [428] := 27.333984, [429] := 27.246094, [430] := 27.070312, [431] := 27.158203, [432] := 25.3125, [433] := 25.40039, [434] := 25.576172, [435] := 25.488281, [436] := 25.927734, [437] := 25.839844, [438] := 25.664062, [439] := 25.751953, [440] := 26.63086, [441] := 26.542969, [442] := 26.367188, [443] := 26.455078, [444] := 26.015625, [445] := 26.103516, [446] := 26.279297, [447] := 26.191406, [448] := 33.66211, [449] := 33.57422, [450] := 33.398438, [451] := 33.48633, [452] := 33.046875, [453] := 33.134766, [454] := 33.310547, [455] := 33.222656, [456] := 32.34375, [457] := 32.43164, [458] := 32.60742, [459] := 32.51953, [460] := 32.958984, [461] := 32.871094, [462] := 32.695312, [463] := 32.783203, [464] := 30.9375, [465] := 31.02539, [466] := 31.201172, [467] := 31.113281, [468] := 31.552734, [469] := 31.464844, [470] := 31.289062, [471] := 31.376953, [472] := 32.25586, [473] := 32.16797, [474] := 31.992188, [475] := 32.08008, [476] := 31.640625, [477] := 31.728516, [478] := 31.904297, [479] := 31.816406, [480] := 28.125,
        [481] := 28.21289, [482] := 28.388672, [483] := 28.300781, [484] := 28.740234, [485] := 28.652344, [486] := 28.476562, [487] := 28.564453, [488] := 29.44336, [489] := 29.355469, [490] := 29.179688, [491] := 29.267578, [492] := 28.828125, [493] := 28.916016, [494] := 29.091797, [495] := 29.003906, [496] := 30.84961, [497] := 30.761719, [498] := 30.585938, [499] := 30.673828, [500] := 30.234375, [501] := 30.322266, [502] := 30.498047, [503] := 30.410156, [504] := 29.53125, [505] := 29.61914, [506] := 29.794922, [507] := 29.707031, [508] := 30.146484, [509] := 30.058594, [510] := 29.882812, [511] := 29.970703, [512] := 89.91211, [513] := 89.82422, [514] := 89.64844, [515] := 89.73633, [516] := 89.296875, [517] := 89.384766, [518] := 89.56055, [519] := 89.47266, [520] := 88.59375, [521] := 88.68164, [522] := 88.85742, [523] := 88.76953, [524] := 89.208984, [525] := 89.12109, [526] := 88.94531, [527] := 89.0332, [528] := 87.1875, [529] := 87.27539, [530] := 87.45117, [531] := 87.36328, [532] := 87.802734, [533] := 87.71484, [534] := 87.53906, [535] := 87.62695, [536] := 88.50586, [537] := 88.41797, [538] := 88.24219, [539] := 88.33008, [540] := 87.890625,
        [541] := 87.978516, [542] := 88.1543, [543] := 88.06641, [544] := 84.375, [545] := 84.46289, [546] := 84.63867, [547] := 84.55078, [548] := 84.990234, [549] := 84.90234, [550] := 84.72656, [551] := 84.81445, [552] := 85.69336, [553] := 85.60547, [554] := 85.42969, [555] := 85.51758, [556] := 85.078125, [557] := 85.166016, [558] := 85.3418, [559] := 85.25391, [560] := 87.09961, [561] := 87.01172, [562] := 86.83594, [563] := 86.92383, [564] := 86.484375, [565] := 86.572266, [566] := 86.74805, [567] := 86.66016, [568] := 85.78125, [569] := 85.86914, [570] := 86.04492, [571] := 85.95703, [572] := 86.396484, [573] := 86.30859, [574] := 86.13281, [575] := 86.2207, [576] := 78.75, [577] := 78.83789, [578] := 79.01367, [579] := 78.92578, [580] := 79.365234, [581] := 79.27734, [582] := 79.10156, [583] := 79.18945, [584] := 80.06836, [585] := 79.98047, [586] := 79.80469, [587] := 79.89258, [588] := 79.453125, [589] := 79.541016, [590] := 79.7168, [591] := 79.62891, [592] := 81.47461, [593] := 81.38672, [594] := 81.21094, [595] := 81.29883, [596] := 80.859375, [597] := 80.947266, [598] := 81.12305, [599] := 81.03516, [600] := 80.15625,
        [601] := 80.24414, [602] := 80.41992, [603] := 80.33203, [604] := 80.771484, [605] := 80.68359, [606] := 80.50781, [607] := 80.5957, [608] := 84.28711, [609] := 84.19922, [610] := 84.02344, [611] := 84.11133, [612] := 83.671875, [613] := 83.759766, [614] := 83.93555, [615] := 83.84766, [616] := 82.96875, [617] := 83.05664, [618] := 83.23242, [619] := 83.14453, [620] := 83.583984, [621] := 83.49609, [622] := 83.32031, [623] := 83.4082, [624] := 81.5625, [625] := 81.65039, [626] := 81.82617, [627] := 81.73828, [628] := 82.177734, [629] := 82.08984, [630] := 81.91406, [631] := 82.00195, [632] := 82.88086, [633] := 82.79297, [634] := 82.61719, [635] := 82.70508, [636] := 82.265625, [637] := 82.353516, [638] := 82.5293, [639] := 82.44141, [640] := 67.5, [641] := 67.58789, [642] := 67.76367, [643] := 67.67578, [644] := 68.115234, [645] := 68.02734, [646] := 67.85156, [647] := 67.93945, [648] := 68.81836, [649] := 68.73047, [650] := 68.55469, [651] := 68.64258, [652] := 68.203125, [653] := 68.291016, [654] := 68.4668, [655] := 68.37891, [656] := 70.22461, [657] := 70.13672, [658] := 69.96094, [659] := 70.04883, [660] := 69.609375,
        [661] := 69.697266, [662] := 69.87305, [663] := 69.78516, [664] := 68.90625, [665] := 68.99414, [666] := 69.16992, [667] := 69.08203, [668] := 69.521484, [669] := 69.43359, [670] := 69.25781, [671] := 69.3457, [672] := 73.03711, [673] := 72.94922, [674] := 72.77344, [675] := 72.86133, [676] := 72.421875, [677] := 72.509766, [678] := 72.68555, [679] := 72.59766, [680] := 71.71875, [681] := 71.80664, [682] := 71.98242, [683] := 71.89453, [684] := 72.333984, [685] := 72.24609, [686] := 72.07031, [687] := 72.1582, [688] := 70.3125, [689] := 70.40039, [690] := 70.57617, [691] := 70.48828, [692] := 70.927734, [693] := 70.83984, [694] := 70.66406, [695] := 70.75195, [696] := 71.63086, [697] := 71.54297, [698] := 71.36719, [699] := 71.45508, [700] := 71.015625, [701] := 71.103516, [702] := 71.2793, [703] := 71.19141, [704] := 78.66211, [705] := 78.57422, [706] := 78.39844, [707] := 78.48633, [708] := 78.046875, [709] := 78.134766, [710] := 78.31055, [711] := 78.22266, [712] := 77.34375, [713] := 77.43164, [714] := 77.60742, [715] := 77.51953, [716] := 77.958984, [717] := 77.87109, [718] := 77.69531, [719] := 77.7832, [720] := 75.9375,
        [721] := 76.02539, [722] := 76.20117, [723] := 76.11328, [724] := 76.552734, [725] := 76.46484, [726] := 76.28906, [727] := 76.37695, [728] := 77.25586, [729] := 77.16797, [730] := 76.99219, [731] := 77.08008, [732] := 76.640625, [733] := 76.728516, [734] := 76.9043, [735] := 76.81641, [736] := 73.125, [737] := 73.21289, [738] := 73.38867, [739] := 73.30078, [740] := 73.740234, [741] := 73.65234, [742] := 73.47656, [743] := 73.56445, [744] := 74.44336, [745] := 74.35547, [746] := 74.17969, [747] := 74.26758, [748] := 73.828125, [749] := 73.916016, [750] := 74.0918, [751] := 74.00391, [752] := 75.84961, [753] := 75.76172, [754] := 75.58594, [755] := 75.67383, [756] := 75.234375, [757] := 75.322266, [758] := 75.49805, [759] := 75.41016, [760] := 74.53125, [761] := 74.61914, [762] := 74.79492, [763] := 74.70703, [764] := 75.146484, [765] := 75.05859, [766] := 74.88281, [767] := 74.9707, [768] := 45.0, [769] := 45.08789, [770] := 45.26367, [771] := 45.17578, [772] := 45.615234, [773] := 45.527344, [774] := 45.351562, [775] := 45.439453, [776] := 46.31836, [777] := 46.23047, [778] := 46.054688, [779] := 46.14258, [780] := 45.703125,
        [781] := 45.791016, [782] := 45.966797, [783] := 45.878906, [784] := 47.72461, [785] := 47.63672, [786] := 47.460938, [787] := 47.54883, [788] := 47.109375, [789] := 47.197266, [790] := 47.373047, [791] := 47.285156, [792] := 46.40625, [793] := 46.49414, [794] := 46.66992, [795] := 46.58203, [796] := 47.021484, [797] := 46.933594, [798] := 46.757812, [799] := 46.845703, [800] := 50.53711, [801] := 50.44922, [802] := 50.273438, [803] := 50.36133, [804] := 49.921875, [805] := 50.009766, [806] := 50.185547, [807] := 50.097656, [808] := 49.21875, [809] := 49.30664, [810] := 49.48242, [811] := 49.39453, [812] := 49.833984, [813] := 49.746094, [814] := 49.570312, [815] := 49.658203, [816] := 47.8125, [817] := 47.90039, [818] := 48.07617, [819] := 47.98828, [820] := 48.427734, [821] := 48.339844, [822] := 48.164062, [823] := 48.251953, [824] := 49.13086, [825] := 49.04297, [826] := 48.867188, [827] := 48.95508, [828] := 48.515625, [829] := 48.603516, [830] := 48.779297, [831] := 48.691406, [832] := 56.16211, [833] := 56.07422, [834] := 55.898438, [835] := 55.98633, [836] := 55.546875, [837] := 55.634766, [838] := 55.810547, [839] := 55.722656, [840] := 54.84375,
        [841] := 54.93164, [842] := 55.10742, [843] := 55.01953, [844] := 55.458984, [845] := 55.371094, [846] := 55.195312, [847] := 55.283203, [848] := 53.4375, [849] := 53.52539, [850] := 53.70117, [851] := 53.61328, [852] := 54.052734, [853] := 53.964844, [854] := 53.789062, [855] := 53.876953, [856] := 54.75586, [857] := 54.66797, [858] := 54.492188, [859] := 54.58008, [860] := 54.140625, [861] := 54.228516, [862] := 54.404297, [863] := 54.316406, [864] := 50.625, [865] := 50.71289, [866] := 50.88867, [867] := 50.80078, [868] := 51.240234, [869] := 51.152344, [870] := 50.976562, [871] := 51.064453, [872] := 51.94336, [873] := 51.85547, [874] := 51.679688, [875] := 51.76758, [876] := 51.328125, [877] := 51.416016, [878] := 51.591797, [879] := 51.503906, [880] := 53.34961, [881] := 53.26172, [882] := 53.085938, [883] := 53.17383, [884] := 52.734375, [885] := 52.822266, [886] := 52.998047, [887] := 52.910156, [888] := 52.03125, [889] := 52.11914, [890] := 52.29492, [891] := 52.20703, [892] := 52.646484, [893] := 52.558594, [894] := 52.382812, [895] := 52.470703, [896] := 67.41211, [897] := 67.32422, [898] := 67.14844, [899] := 67.23633, [900] := 66.796875,
        [901] := 66.884766, [902] := 67.06055, [903] := 66.97266, [904] := 66.09375, [905] := 66.18164, [906] := 66.35742, [907] := 66.26953, [908] := 66.708984, [909] := 66.62109, [910] := 66.44531, [911] := 66.5332, [912] := 64.6875, [913] := 64.77539, [914] := 64.95117, [915] := 64.86328, [916] := 65.302734, [917] := 65.21484, [918] := 65.03906, [919] := 65.12695, [920] := 66.00586, [921] := 65.91797, [922] := 65.74219, [923] := 65.83008, [924] := 65.390625, [925] := 65.478516, [926] := 65.6543, [927] := 65.56641, [928] := 61.875, [929] := 61.96289, [930] := 62.13867, [931] := 62.05078, [932] := 62.490234, [933] := 62.402344, [934] := 62.226562, [935] := 62.314453, [936] := 63.19336, [937] := 63.10547, [938] := 62.929688, [939] := 63.01758, [940] := 62.578125, [941] := 62.666016, [942] := 62.841797, [943] := 62.753906, [944] := 64.59961, [945] := 64.51172, [946] := 64.33594, [947] := 64.42383, [948] := 63.984375, [949] := 64.072266, [950] := 64.24805, [951] := 64.16016, [952] := 63.28125, [953] := 63.36914, [954] := 63.54492, [955] := 63.45703, [956] := 63.896484, [957] := 63.808594, [958] := 63.632812, [959] := 63.720703, [960] := 56.25,
        [961] := 56.33789, [962] := 56.51367, [963] := 56.42578, [964] := 56.865234, [965] := 56.777344, [966] := 56.601562, [967] := 56.689453, [968] := 57.56836, [969] := 57.48047, [970] := 57.304688, [971] := 57.39258, [972] := 56.953125, [973] := 57.041016, [974] := 57.216797, [975] := 57.128906, [976] := 58.97461, [977] := 58.88672, [978] := 58.710938, [979] := 58.79883, [980] := 58.359375, [981] := 58.447266, [982] := 58.623047, [983] := 58.535156, [984] := 57.65625, [985] := 57.74414, [986] := 57.91992, [987] := 57.83203, [988] := 58.271484, [989] := 58.183594, [990] := 58.007812, [991] := 58.095703, [992] := 61.78711, [993] := 61.69922, [994] := 61.523438, [995] := 61.61133, [996] := 61.171875, [997] := 61.259766, [998] := 61.435547, [999] := 61.347656, [1000] := 60.46875, [1001] := 60.55664, [1002] := 60.73242, [1003] := 60.64453, [1004] := 61.083984, [1005] := 60.996094, [1006] := 60.820312, [1007] := 60.908203, [1008] := 59.0625, [1009] := 59.15039, [1010] := 59.32617, [1011] := 59.23828, [1012] := 59.677734, [1013] := 59.589844, [1014] := 59.414062, [1015] := 59.501953, [1016] := 60.38086, [1017] := 60.29297, [1018] := 60.117188, [1019] := 60.20508, [1020] := 59.765625,
        [1021] := 59.853516, [1022] := 60.029297, [1023] := 59.941406, [1024] := 179.91211, [1025] := 179.82422, [1026] := 179.64844, [1027] := 179.73633, [1028] := 179.29688, [1029] := 179.38477, [1030] := 179.56055, [1031] := 179.47266, [1032] := 178.59375, [1033] := 178.68164, [1034] := 178.85742, [1035] := 178.76953, [1036] := 179.20898, [1037] := 179.1211, [1038] := 178.94531, [1039] := 179.0332, [1040] := 177.1875, [1041] := 177.27539, [1042] := 177.45117, [1043] := 177.36328, [1044] := 177.80273, [1045] := 177.71484, [1046] := 177.53906, [1047] := 177.62695, [1048] := 178.50586, [1049] := 178.41797, [1050] := 178.24219, [1051] := 178.33008, [1052] := 177.89062, [1053] := 177.97852, [1054] := 178.1543, [1055] := 178.0664, [1056] := 174.375, [1057] := 174.46289, [1058] := 174.63867, [1059] := 174.55078, [1060] := 174.99023, [1061] := 174.90234, [1062] := 174.72656, [1063] := 174.81445, [1064] := 175.69336, [1065] := 175.60547, [1066] := 175.42969, [1067] := 175.51758, [1068] := 175.07812, [1069] := 175.16602, [1070] := 175.3418, [1071] := 175.2539, [1072] := 177.09961, [1073] := 177.01172, [1074] := 176.83594, [1075] := 176.92383, [1076] := 176.48438, [1077] := 176.57227, [1078] := 176.74805, [1079] := 176.66016, [1080] := 175.78125,
        [1081] := 175.86914, [1082] := 176.04492, [1083] := 175.95703, [1084] := 176.39648, [1085] := 176.3086, [1086] := 176.13281, [1087] := 176.2207, [1088] := 168.75, [1089] := 168.83789, [1090] := 169.01367, [1091] := 168.92578, [1092] := 169.36523, [1093] := 169.27734, [1094] := 169.10156, [1095] := 169.18945, [1096] := 170.06836, [1097] := 169.98047, [1098] := 169.80469, [1099] := 169.89258, [1100] := 169.45312, [1101] := 169.54102, [1102] := 169.7168, [1103] := 169.6289, [1104] := 171.47461, [1105] := 171.38672, [1106] := 171.21094, [1107] := 171.29883, [1108] := 170.85938, [1109] := 170.94727, [1110] := 171.12305, [1111] := 171.03516, [1112] := 170.15625, [1113] := 170.24414, [1114] := 170.41992, [1115] := 170.33203, [1116] := 170.77148, [1117] := 170.6836, [1118] := 170.50781, [1119] := 170.5957, [1120] := 174.28711, [1121] := 174.19922, [1122] := 174.02344, [1123] := 174.11133, [1124] := 173.67188, [1125] := 173.75977, [1126] := 173.93555, [1127] := 173.84766, [1128] := 172.96875, [1129] := 173.05664, [1130] := 173.23242, [1131] := 173.14453, [1132] := 173.58398, [1133] := 173.4961, [1134] := 173.32031, [1135] := 173.4082, [1136] := 171.5625, [1137] := 171.65039, [1138] := 171.82617, [1139] := 171.73828, [1140] := 172.17773,
        [1141] := 172.08984, [1142] := 171.91406, [1143] := 172.00195, [1144] := 172.88086, [1145] := 172.79297, [1146] := 172.61719, [1147] := 172.70508, [1148] := 172.26562, [1149] := 172.35352, [1150] := 172.5293, [1151] := 172.4414, [1152] := 157.5, [1153] := 157.58789, [1154] := 157.76367, [1155] := 157.67578, [1156] := 158.11523, [1157] := 158.02734, [1158] := 157.85156, [1159] := 157.93945, [1160] := 158.81836, [1161] := 158.73047, [1162] := 158.55469, [1163] := 158.64258, [1164] := 158.20312, [1165] := 158.29102, [1166] := 158.4668, [1167] := 158.3789, [1168] := 160.22461, [1169] := 160.13672, [1170] := 159.96094, [1171] := 160.04883, [1172] := 159.60938, [1173] := 159.69727, [1174] := 159.87305, [1175] := 159.78516, [1176] := 158.90625, [1177] := 158.99414, [1178] := 159.16992, [1179] := 159.08203, [1180] := 159.52148, [1181] := 159.4336, [1182] := 159.25781, [1183] := 159.3457, [1184] := 163.03711, [1185] := 162.94922, [1186] := 162.77344, [1187] := 162.86133, [1188] := 162.42188, [1189] := 162.50977, [1190] := 162.68555, [1191] := 162.59766, [1192] := 161.71875, [1193] := 161.80664, [1194] := 161.98242, [1195] := 161.89453, [1196] := 162.33398, [1197] := 162.2461, [1198] := 162.07031, [1199] := 162.1582, [1200] := 160.3125,
        [1201] := 160.40039, [1202] := 160.57617, [1203] := 160.48828, [1204] := 160.92773, [1205] := 160.83984, [1206] := 160.66406, [1207] := 160.75195, [1208] := 161.63086, [1209] := 161.54297, [1210] := 161.36719, [1211] := 161.45508, [1212] := 161.01562, [1213] := 161.10352, [1214] := 161.2793, [1215] := 161.1914, [1216] := 168.66211, [1217] := 168.57422, [1218] := 168.39844, [1219] := 168.48633, [1220] := 168.04688, [1221] := 168.13477, [1222] := 168.31055, [1223] := 168.22266, [1224] := 167.34375, [1225] := 167.43164, [1226] := 167.60742, [1227] := 167.51953, [1228] := 167.95898, [1229] := 167.8711, [1230] := 167.69531, [1231] := 167.7832, [1232] := 165.9375, [1233] := 166.02539, [1234] := 166.20117, [1235] := 166.11328, [1236] := 166.55273, [1237] := 166.46484, [1238] := 166.28906, [1239] := 166.37695, [1240] := 167.25586, [1241] := 167.16797, [1242] := 166.99219, [1243] := 167.08008, [1244] := 166.64062, [1245] := 166.72852, [1246] := 166.9043, [1247] := 166.8164, [1248] := 163.125, [1249] := 163.21289, [1250] := 163.38867, [1251] := 163.30078, [1252] := 163.74023, [1253] := 163.65234, [1254] := 163.47656, [1255] := 163.56445, [1256] := 164.44336, [1257] := 164.35547, [1258] := 164.17969, [1259] := 164.26758, [1260] := 163.82812,
        [1261] := 163.91602, [1262] := 164.0918, [1263] := 164.0039, [1264] := 165.84961, [1265] := 165.76172, [1266] := 165.58594, [1267] := 165.67383, [1268] := 165.23438, [1269] := 165.32227, [1270] := 165.49805, [1271] := 165.41016, [1272] := 164.53125, [1273] := 164.61914, [1274] := 164.79492, [1275] := 164.70703, [1276] := 165.14648, [1277] := 165.0586, [1278] := 164.88281, [1279] := 164.9707, [1280] := 135.0, [1281] := 135.08789, [1282] := 135.26367, [1283] := 135.17578, [1284] := 135.61523, [1285] := 135.52734, [1286] := 135.35156, [1287] := 135.43945, [1288] := 136.31836, [1289] := 136.23047, [1290] := 136.05469, [1291] := 136.14258, [1292] := 135.70312, [1293] := 135.79102, [1294] := 135.9668, [1295] := 135.8789, [1296] := 137.72461, [1297] := 137.63672, [1298] := 137.46094, [1299] := 137.54883, [1300] := 137.10938, [1301] := 137.19727, [1302] := 137.37305, [1303] := 137.28516, [1304] := 136.40625, [1305] := 136.49414, [1306] := 136.66992, [1307] := 136.58203, [1308] := 137.02148, [1309] := 136.9336, [1310] := 136.75781, [1311] := 136.8457, [1312] := 140.53711, [1313] := 140.44922, [1314] := 140.27344, [1315] := 140.36133, [1316] := 139.92188, [1317] := 140.00977, [1318] := 140.18555, [1319] := 140.09766, [1320] := 139.21875,
        [1321] := 139.30664, [1322] := 139.48242, [1323] := 139.39453, [1324] := 139.83398, [1325] := 139.7461, [1326] := 139.57031, [1327] := 139.6582, [1328] := 137.8125, [1329] := 137.90039, [1330] := 138.07617, [1331] := 137.98828, [1332] := 138.42773, [1333] := 138.33984, [1334] := 138.16406, [1335] := 138.25195, [1336] := 139.13086, [1337] := 139.04297, [1338] := 138.86719, [1339] := 138.95508, [1340] := 138.51562, [1341] := 138.60352, [1342] := 138.7793, [1343] := 138.6914, [1344] := 146.16211, [1345] := 146.07422, [1346] := 145.89844, [1347] := 145.98633, [1348] := 145.54688, [1349] := 145.63477, [1350] := 145.81055, [1351] := 145.72266, [1352] := 144.84375, [1353] := 144.93164, [1354] := 145.10742, [1355] := 145.01953, [1356] := 145.45898, [1357] := 145.3711, [1358] := 145.19531, [1359] := 145.2832, [1360] := 143.4375, [1361] := 143.52539, [1362] := 143.70117, [1363] := 143.61328, [1364] := 144.05273, [1365] := 143.96484, [1366] := 143.78906, [1367] := 143.87695, [1368] := 144.75586, [1369] := 144.66797, [1370] := 144.49219, [1371] := 144.58008, [1372] := 144.14062, [1373] := 144.22852, [1374] := 144.4043, [1375] := 144.3164, [1376] := 140.625, [1377] := 140.71289, [1378] := 140.88867, [1379] := 140.80078, [1380] := 141.24023,
        [1381] := 141.15234, [1382] := 140.97656, [1383] := 141.06445, [1384] := 141.94336, [1385] := 141.85547, [1386] := 141.67969, [1387] := 141.76758, [1388] := 141.32812, [1389] := 141.41602, [1390] := 141.5918, [1391] := 141.5039, [1392] := 143.34961, [1393] := 143.26172, [1394] := 143.08594, [1395] := 143.17383, [1396] := 142.73438, [1397] := 142.82227, [1398] := 142.99805, [1399] := 142.91016, [1400] := 142.03125, [1401] := 142.11914, [1402] := 142.29492, [1403] := 142.20703, [1404] := 142.64648, [1405] := 142.5586, [1406] := 142.38281, [1407] := 142.4707, [1408] := 157.41211, [1409] := 157.32422, [1410] := 157.14844, [1411] := 157.23633, [1412] := 156.79688, [1413] := 156.88477, [1414] := 157.06055, [1415] := 156.97266, [1416] := 156.09375, [1417] := 156.18164, [1418] := 156.35742, [1419] := 156.26953, [1420] := 156.70898, [1421] := 156.6211, [1422] := 156.44531, [1423] := 156.5332, [1424] := 154.6875, [1425] := 154.77539, [1426] := 154.95117, [1427] := 154.86328, [1428] := 155.30273, [1429] := 155.21484, [1430] := 155.03906, [1431] := 155.12695, [1432] := 156.00586, [1433] := 155.91797, [1434] := 155.74219, [1435] := 155.83008, [1436] := 155.39062, [1437] := 155.47852, [1438] := 155.6543, [1439] := 155.5664, [1440] := 151.875,
        [1441] := 151.96289, [1442] := 152.13867, [1443] := 152.05078, [1444] := 152.49023, [1445] := 152.40234, [1446] := 152.22656, [1447] := 152.31445, [1448] := 153.19336, [1449] := 153.10547, [1450] := 152.92969, [1451] := 153.01758, [1452] := 152.57812, [1453] := 152.66602, [1454] := 152.8418, [1455] := 152.7539, [1456] := 154.59961, [1457] := 154.51172, [1458] := 154.33594, [1459] := 154.42383, [1460] := 153.98438, [1461] := 154.07227, [1462] := 154.24805, [1463] := 154.16016, [1464] := 153.28125, [1465] := 153.36914, [1466] := 153.54492, [1467] := 153.45703, [1468] := 153.89648, [1469] := 153.8086, [1470] := 153.63281, [1471] := 153.7207, [1472] := 146.25, [1473] := 146.33789, [1474] := 146.51367, [1475] := 146.42578, [1476] := 146.86523, [1477] := 146.77734, [1478] := 146.60156, [1479] := 146.68945, [1480] := 147.56836, [1481] := 147.48047, [1482] := 147.30469, [1483] := 147.39258, [1484] := 146.95312, [1485] := 147.04102, [1486] := 147.2168, [1487] := 147.1289, [1488] := 148.97461, [1489] := 148.88672, [1490] := 148.71094, [1491] := 148.79883, [1492] := 148.35938, [1493] := 148.44727, [1494] := 148.62305, [1495] := 148.53516, [1496] := 147.65625, [1497] := 147.74414, [1498] := 147.91992, [1499] := 147.83203, [1500] := 148.27148,
        [1501] := 148.1836, [1502] := 148.00781, [1503] := 148.0957, [1504] := 151.78711, [1505] := 151.69922, [1506] := 151.52344, [1507] := 151.61133, [1508] := 151.17188, [1509] := 151.25977, [1510] := 151.43555, [1511] := 151.34766, [1512] := 150.46875, [1513] := 150.55664, [1514] := 150.73242, [1515] := 150.64453, [1516] := 151.08398, [1517] := 150.9961, [1518] := 150.82031, [1519] := 150.9082, [1520] := 149.0625, [1521] := 149.15039, [1522] := 149.32617, [1523] := 149.23828, [1524] := 149.67773, [1525] := 149.58984, [1526] := 149.41406, [1527] := 149.50195, [1528] := 150.38086, [1529] := 150.29297, [1530] := 150.11719, [1531] := 150.20508, [1532] := 149.76562, [1533] := 149.85352, [1534] := 150.0293, [1535] := 149.9414, [1536] := 90.0, [1537] := 90.08789, [1538] := 90.26367, [1539] := 90.17578, [1540] := 90.615234, [1541] := 90.52734, [1542] := 90.35156, [1543] := 90.43945, [1544] := 91.31836, [1545] := 91.23047, [1546] := 91.05469, [1547] := 91.14258, [1548] := 90.703125, [1549] := 90.791016, [1550] := 90.9668, [1551] := 90.87891, [1552] := 92.72461, [1553] := 92.63672, [1554] := 92.46094, [1555] := 92.54883, [1556] := 92.109375, [1557] := 92.197266, [1558] := 92.37305, [1559] := 92.28516, [1560] := 91.40625,
        [1561] := 91.49414, [1562] := 91.66992, [1563] := 91.58203, [1564] := 92.021484, [1565] := 91.93359, [1566] := 91.75781, [1567] := 91.8457, [1568] := 95.53711, [1569] := 95.44922, [1570] := 95.27344, [1571] := 95.36133, [1572] := 94.921875, [1573] := 95.009766, [1574] := 95.18555, [1575] := 95.09766, [1576] := 94.21875, [1577] := 94.30664, [1578] := 94.48242, [1579] := 94.39453, [1580] := 94.833984, [1581] := 94.74609, [1582] := 94.57031, [1583] := 94.6582, [1584] := 92.8125, [1585] := 92.90039, [1586] := 93.07617, [1587] := 92.98828, [1588] := 93.427734, [1589] := 93.33984, [1590] := 93.16406, [1591] := 93.25195, [1592] := 94.13086, [1593] := 94.04297, [1594] := 93.86719, [1595] := 93.95508, [1596] := 93.515625, [1597] := 93.603516, [1598] := 93.7793, [1599] := 93.69141, [1600] := 101.16211, [1601] := 101.07422, [1602] := 100.89844, [1603] := 100.98633, [1604] := 100.546875, [1605] := 100.634766, [1606] := 100.81055, [1607] := 100.72266, [1608] := 99.84375, [1609] := 99.93164, [1610] := 100.10742, [1611] := 100.01953, [1612] := 100.458984, [1613] := 100.37109, [1614] := 100.19531, [1615] := 100.2832, [1616] := 98.4375, [1617] := 98.52539, [1618] := 98.70117, [1619] := 98.61328, [1620] := 99.052734,
        [1621] := 98.96484, [1622] := 98.78906, [1623] := 98.87695, [1624] := 99.75586, [1625] := 99.66797, [1626] := 99.49219, [1627] := 99.58008, [1628] := 99.140625, [1629] := 99.228516, [1630] := 99.4043, [1631] := 99.31641, [1632] := 95.625, [1633] := 95.71289, [1634] := 95.88867, [1635] := 95.80078, [1636] := 96.240234, [1637] := 96.15234, [1638] := 95.97656, [1639] := 96.06445, [1640] := 96.94336, [1641] := 96.85547, [1642] := 96.67969, [1643] := 96.76758, [1644] := 96.328125, [1645] := 96.416016, [1646] := 96.5918, [1647] := 96.50391, [1648] := 98.34961, [1649] := 98.26172, [1650] := 98.08594, [1651] := 98.17383, [1652] := 97.734375, [1653] := 97.822266, [1654] := 97.99805, [1655] := 97.91016, [1656] := 97.03125, [1657] := 97.11914, [1658] := 97.29492, [1659] := 97.20703, [1660] := 97.646484, [1661] := 97.55859, [1662] := 97.38281, [1663] := 97.4707, [1664] := 112.41211, [1665] := 112.32422, [1666] := 112.14844, [1667] := 112.23633, [1668] := 111.796875, [1669] := 111.884766, [1670] := 112.06055, [1671] := 111.97266, [1672] := 111.09375, [1673] := 111.18164, [1674] := 111.35742, [1675] := 111.26953, [1676] := 111.708984, [1677] := 111.62109, [1678] := 111.44531, [1679] := 111.5332, [1680] := 109.6875,
        [1681] := 109.77539, [1682] := 109.95117, [1683] := 109.86328, [1684] := 110.302734, [1685] := 110.21484, [1686] := 110.03906, [1687] := 110.12695, [1688] := 111.00586, [1689] := 110.91797, [1690] := 110.74219, [1691] := 110.83008, [1692] := 110.390625, [1693] := 110.478516, [1694] := 110.6543, [1695] := 110.56641, [1696] := 106.875, [1697] := 106.96289, [1698] := 107.13867, [1699] := 107.05078, [1700] := 107.490234, [1701] := 107.40234, [1702] := 107.22656, [1703] := 107.31445, [1704] := 108.19336, [1705] := 108.10547, [1706] := 107.92969, [1707] := 108.01758, [1708] := 107.578125, [1709] := 107.666016, [1710] := 107.8418, [1711] := 107.75391, [1712] := 109.59961, [1713] := 109.51172, [1714] := 109.33594, [1715] := 109.42383, [1716] := 108.984375, [1717] := 109.072266, [1718] := 109.24805, [1719] := 109.16016, [1720] := 108.28125, [1721] := 108.36914, [1722] := 108.54492, [1723] := 108.45703, [1724] := 108.896484, [1725] := 108.80859, [1726] := 108.63281, [1727] := 108.7207, [1728] := 101.25, [1729] := 101.33789, [1730] := 101.51367, [1731] := 101.42578, [1732] := 101.865234, [1733] := 101.77734, [1734] := 101.60156, [1735] := 101.68945, [1736] := 102.56836, [1737] := 102.48047, [1738] := 102.30469, [1739] := 102.39258, [1740] := 101.953125,
        [1741] := 102.041016, [1742] := 102.2168, [1743] := 102.12891, [1744] := 103.97461, [1745] := 103.88672, [1746] := 103.71094, [1747] := 103.79883, [1748] := 103.359375, [1749] := 103.447266, [1750] := 103.62305, [1751] := 103.53516, [1752] := 102.65625, [1753] := 102.74414, [1754] := 102.91992, [1755] := 102.83203, [1756] := 103.271484, [1757] := 103.18359, [1758] := 103.00781, [1759] := 103.0957, [1760] := 106.78711, [1761] := 106.69922, [1762] := 106.52344, [1763] := 106.61133, [1764] := 106.171875, [1765] := 106.259766, [1766] := 106.43555, [1767] := 106.34766, [1768] := 105.46875, [1769] := 105.55664, [1770] := 105.73242, [1771] := 105.64453, [1772] := 106.083984, [1773] := 105.99609, [1774] := 105.82031, [1775] := 105.9082, [1776] := 104.0625, [1777] := 104.15039, [1778] := 104.32617, [1779] := 104.23828, [1780] := 104.677734, [1781] := 104.58984, [1782] := 104.41406, [1783] := 104.50195, [1784] := 105.38086, [1785] := 105.29297, [1786] := 105.11719, [1787] := 105.20508, [1788] := 104.765625, [1789] := 104.853516, [1790] := 105.0293, [1791] := 104.94141, [1792] := 134.91211, [1793] := 134.82422, [1794] := 134.64844, [1795] := 134.73633, [1796] := 134.29688, [1797] := 134.38477, [1798] := 134.56055, [1799] := 134.47266, [1800] := 133.59375,
        [1801] := 133.68164, [1802] := 133.85742, [1803] := 133.76953, [1804] := 134.20898, [1805] := 134.1211, [1806] := 133.94531, [1807] := 134.0332, [1808] := 132.1875, [1809] := 132.27539, [1810] := 132.45117, [1811] := 132.36328, [1812] := 132.80273, [1813] := 132.71484, [1814] := 132.53906, [1815] := 132.62695, [1816] := 133.50586, [1817] := 133.41797, [1818] := 133.24219, [1819] := 133.33008, [1820] := 132.89062, [1821] := 132.97852, [1822] := 133.1543, [1823] := 133.0664, [1824] := 129.375, [1825] := 129.46289, [1826] := 129.63867, [1827] := 129.55078, [1828] := 129.99023, [1829] := 129.90234, [1830] := 129.72656, [1831] := 129.81445, [1832] := 130.69336, [1833] := 130.60547, [1834] := 130.42969, [1835] := 130.51758, [1836] := 130.07812, [1837] := 130.16602, [1838] := 130.3418, [1839] := 130.2539, [1840] := 132.09961, [1841] := 132.01172, [1842] := 131.83594, [1843] := 131.92383, [1844] := 131.48438, [1845] := 131.57227, [1846] := 131.74805, [1847] := 131.66016, [1848] := 130.78125, [1849] := 130.86914, [1850] := 131.04492, [1851] := 130.95703, [1852] := 131.39648, [1853] := 131.3086, [1854] := 131.13281, [1855] := 131.2207, [1856] := 123.75, [1857] := 123.83789, [1858] := 124.01367, [1859] := 123.92578, [1860] := 124.365234,
        [1861] := 124.27734, [1862] := 124.10156, [1863] := 124.18945, [1864] := 125.06836, [1865] := 124.98047, [1866] := 124.80469, [1867] := 124.89258, [1868] := 124.453125, [1869] := 124.541016, [1870] := 124.7168, [1871] := 124.62891, [1872] := 126.47461, [1873] := 126.38672, [1874] := 126.21094, [1875] := 126.29883, [1876] := 125.859375, [1877] := 125.947266, [1878] := 126.12305, [1879] := 126.03516, [1880] := 125.15625, [1881] := 125.24414, [1882] := 125.41992, [1883] := 125.33203, [1884] := 125.771484, [1885] := 125.68359, [1886] := 125.50781, [1887] := 125.5957, [1888] := 129.28711, [1889] := 129.19922, [1890] := 129.02344, [1891] := 129.11133, [1892] := 128.67188, [1893] := 128.75977, [1894] := 128.93555, [1895] := 128.84766, [1896] := 127.96875, [1897] := 128.05664, [1898] := 128.23242, [1899] := 128.14453, [1900] := 128.58398, [1901] := 128.4961, [1902] := 128.32031, [1903] := 128.4082, [1904] := 126.5625, [1905] := 126.65039, [1906] := 126.82617, [1907] := 126.73828, [1908] := 127.177734, [1909] := 127.08984, [1910] := 126.91406, [1911] := 127.00195, [1912] := 127.88086, [1913] := 127.79297, [1914] := 127.61719, [1915] := 127.70508, [1916] := 127.265625, [1917] := 127.353516, [1918] := 127.5293, [1919] := 127.44141, [1920] := 112.5,
        [1921] := 112.58789, [1922] := 112.76367, [1923] := 112.67578, [1924] := 113.115234, [1925] := 113.02734, [1926] := 112.85156, [1927] := 112.93945, [1928] := 113.81836, [1929] := 113.73047, [1930] := 113.55469, [1931] := 113.64258, [1932] := 113.203125, [1933] := 113.291016, [1934] := 113.4668, [1935] := 113.37891, [1936] := 115.22461, [1937] := 115.13672, [1938] := 114.96094, [1939] := 115.04883, [1940] := 114.609375, [1941] := 114.697266, [1942] := 114.87305, [1943] := 114.78516, [1944] := 113.90625, [1945] := 113.99414, [1946] := 114.16992, [1947] := 114.08203, [1948] := 114.521484, [1949] := 114.43359, [1950] := 114.25781, [1951] := 114.3457, [1952] := 118.03711, [1953] := 117.94922, [1954] := 117.77344, [1955] := 117.86133, [1956] := 117.421875, [1957] := 117.509766, [1958] := 117.68555, [1959] := 117.59766, [1960] := 116.71875, [1961] := 116.80664, [1962] := 116.98242, [1963] := 116.89453, [1964] := 117.333984, [1965] := 117.24609, [1966] := 117.07031, [1967] := 117.1582, [1968] := 115.3125, [1969] := 115.40039, [1970] := 115.57617, [1971] := 115.48828, [1972] := 115.927734, [1973] := 115.83984, [1974] := 115.66406, [1975] := 115.75195, [1976] := 116.63086, [1977] := 116.54297, [1978] := 116.36719, [1979] := 116.45508, [1980] := 116.015625,
        [1981] := 116.103516, [1982] := 116.2793, [1983] := 116.19141, [1984] := 123.66211, [1985] := 123.57422, [1986] := 123.39844, [1987] := 123.48633, [1988] := 123.046875, [1989] := 123.134766, [1990] := 123.31055, [1991] := 123.22266, [1992] := 122.34375, [1993] := 122.43164, [1994] := 122.60742, [1995] := 122.51953, [1996] := 122.958984, [1997] := 122.87109, [1998] := 122.69531, [1999] := 122.7832, [2000] := 120.9375, [2001] := 121.02539, [2002] := 121.20117, [2003] := 121.11328, [2004] := 121.552734, [2005] := 121.46484, [2006] := 121.28906, [2007] := 121.37695, [2008] := 122.25586, [2009] := 122.16797, [2010] := 121.99219, [2011] := 122.08008, [2012] := 121.640625, [2013] := 121.728516, [2014] := 121.9043, [2015] := 121.81641, [2016] := 118.125, [2017] := 118.21289, [2018] := 118.38867, [2019] := 118.30078, [2020] := 118.740234, [2021] := 118.65234, [2022] := 118.47656, [2023] := 118.56445, [2024] := 119.44336, [2025] := 119.35547, [2026] := 119.17969, [2027] := 119.26758, [2028] := 118.828125, [2029] := 118.916016, [2030] := 119.0918, [2031] := 119.00391, [2032] := 120.84961, [2033] := 120.76172, [2034] := 120.58594, [2035] := 120.67383, [2036] := 120.234375, [2037] := 120.322266, [2038] := 120.49805, [2039] := 120.41016, [2040] := 119.53125,
        [2041] := 119.61914, [2042] := 119.79492, [2043] := 119.70703, [2044] := 120.146484, [2045] := 120.05859, [2046] := 119.88281, [2047] := 119.9707, [2048] := 359.9121, [2049] := 359.82422, [2050] := 359.64844, [2051] := 359.73633, [2052] := 359.29688, [2053] := 359.38477, [2054] := 359.56055, [2055] := 359.47266, [2056] := 358.59375, [2057] := 358.68164, [2058] := 358.85742, [2059] := 358.76953, [2060] := 359.20898, [2061] := 359.1211, [2062] := 358.9453, [2063] := 359.0332, [2064] := 357.1875, [2065] := 357.2754, [2066] := 357.45117, [2067] := 357.36328, [2068] := 357.80273, [2069] := 357.71484, [2070] := 357.53906, [2071] := 357.62695, [2072] := 358.50586, [2073] := 358.41797, [2074] := 358.2422, [2075] := 358.33008, [2076] := 357.89062, [2077] := 357.97852, [2078] := 358.1543, [2079] := 358.0664, [2080] := 354.375, [2081] := 354.4629, [2082] := 354.63867, [2083] := 354.55078, [2084] := 354.99023, [2085] := 354.90234, [2086] := 354.72656, [2087] := 354.81445, [2088] := 355.69336, [2089] := 355.60547, [2090] := 355.4297, [2091] := 355.51758, [2092] := 355.07812, [2093] := 355.16602, [2094] := 355.3418, [2095] := 355.2539, [2096] := 357.0996, [2097] := 357.01172, [2098] := 356.83594, [2099] := 356.92383, [2100] := 356.48438,
        [2101] := 356.57227, [2102] := 356.74805, [2103] := 356.66016, [2104] := 355.78125, [2105] := 355.86914, [2106] := 356.04492, [2107] := 355.95703, [2108] := 356.39648, [2109] := 356.3086, [2110] := 356.1328, [2111] := 356.2207, [2112] := 348.75, [2113] := 348.8379, [2114] := 349.01367, [2115] := 348.92578, [2116] := 349.36523, [2117] := 349.27734, [2118] := 349.10156, [2119] := 349.18945, [2120] := 350.06836, [2121] := 349.98047, [2122] := 349.8047, [2123] := 349.89258, [2124] := 349.45312, [2125] := 349.54102, [2126] := 349.7168, [2127] := 349.6289, [2128] := 351.4746, [2129] := 351.38672, [2130] := 351.21094, [2131] := 351.29883, [2132] := 350.85938, [2133] := 350.94727, [2134] := 351.12305, [2135] := 351.03516, [2136] := 350.15625, [2137] := 350.24414, [2138] := 350.41992, [2139] := 350.33203, [2140] := 350.77148, [2141] := 350.6836, [2142] := 350.5078, [2143] := 350.5957, [2144] := 354.2871, [2145] := 354.19922, [2146] := 354.02344, [2147] := 354.11133, [2148] := 353.67188, [2149] := 353.75977, [2150] := 353.93555, [2151] := 353.84766, [2152] := 352.96875, [2153] := 353.05664, [2154] := 353.23242, [2155] := 353.14453, [2156] := 353.58398, [2157] := 353.4961, [2158] := 353.3203, [2159] := 353.4082, [2160] := 351.5625,
        [2161] := 351.6504, [2162] := 351.82617, [2163] := 351.73828, [2164] := 352.17773, [2165] := 352.08984, [2166] := 351.91406, [2167] := 352.00195, [2168] := 352.88086, [2169] := 352.79297, [2170] := 352.6172, [2171] := 352.70508, [2172] := 352.26562, [2173] := 352.35352, [2174] := 352.5293, [2175] := 352.4414, [2176] := 337.5, [2177] := 337.5879, [2178] := 337.76367, [2179] := 337.67578, [2180] := 338.11523, [2181] := 338.02734, [2182] := 337.85156, [2183] := 337.93945, [2184] := 338.81836, [2185] := 338.73047, [2186] := 338.5547, [2187] := 338.64258, [2188] := 338.20312, [2189] := 338.29102, [2190] := 338.4668, [2191] := 338.3789, [2192] := 340.2246, [2193] := 340.13672, [2194] := 339.96094, [2195] := 340.04883, [2196] := 339.60938, [2197] := 339.69727, [2198] := 339.87305, [2199] := 339.78516, [2200] := 338.90625, [2201] := 338.99414, [2202] := 339.16992, [2203] := 339.08203, [2204] := 339.52148, [2205] := 339.4336, [2206] := 339.2578, [2207] := 339.3457, [2208] := 343.0371, [2209] := 342.94922, [2210] := 342.77344, [2211] := 342.86133, [2212] := 342.42188, [2213] := 342.50977, [2214] := 342.68555, [2215] := 342.59766, [2216] := 341.71875, [2217] := 341.80664, [2218] := 341.98242, [2219] := 341.89453, [2220] := 342.33398,
        [2221] := 342.2461, [2222] := 342.0703, [2223] := 342.1582, [2224] := 340.3125, [2225] := 340.4004, [2226] := 340.57617, [2227] := 340.48828, [2228] := 340.92773, [2229] := 340.83984, [2230] := 340.66406, [2231] := 340.75195, [2232] := 341.63086, [2233] := 341.54297, [2234] := 341.3672, [2235] := 341.45508, [2236] := 341.01562, [2237] := 341.10352, [2238] := 341.2793, [2239] := 341.1914, [2240] := 348.6621, [2241] := 348.57422, [2242] := 348.39844, [2243] := 348.48633, [2244] := 348.04688, [2245] := 348.13477, [2246] := 348.31055, [2247] := 348.22266, [2248] := 347.34375, [2249] := 347.43164, [2250] := 347.60742, [2251] := 347.51953, [2252] := 347.95898, [2253] := 347.8711, [2254] := 347.6953, [2255] := 347.7832, [2256] := 345.9375, [2257] := 346.0254, [2258] := 346.20117, [2259] := 346.11328, [2260] := 346.55273, [2261] := 346.46484, [2262] := 346.28906, [2263] := 346.37695, [2264] := 347.25586, [2265] := 347.16797, [2266] := 346.9922, [2267] := 347.08008, [2268] := 346.64062, [2269] := 346.72852, [2270] := 346.9043, [2271] := 346.8164, [2272] := 343.125, [2273] := 343.2129, [2274] := 343.38867, [2275] := 343.30078, [2276] := 343.74023, [2277] := 343.65234, [2278] := 343.47656, [2279] := 343.56445, [2280] := 344.44336,
        [2281] := 344.35547, [2282] := 344.1797, [2283] := 344.26758, [2284] := 343.82812, [2285] := 343.91602, [2286] := 344.0918, [2287] := 344.0039, [2288] := 345.8496, [2289] := 345.76172, [2290] := 345.58594, [2291] := 345.67383, [2292] := 345.23438, [2293] := 345.32227, [2294] := 345.49805, [2295] := 345.41016, [2296] := 344.53125, [2297] := 344.61914, [2298] := 344.79492, [2299] := 344.70703, [2300] := 345.14648, [2301] := 345.0586, [2302] := 344.8828, [2303] := 344.9707, [2304] := 315.0, [2305] := 315.0879, [2306] := 315.26367, [2307] := 315.17578, [2308] := 315.61523, [2309] := 315.52734, [2310] := 315.35156, [2311] := 315.43945, [2312] := 316.31836, [2313] := 316.23047, [2314] := 316.0547, [2315] := 316.14258, [2316] := 315.70312, [2317] := 315.79102, [2318] := 315.9668, [2319] := 315.8789, [2320] := 317.7246, [2321] := 317.63672, [2322] := 317.46094, [2323] := 317.54883, [2324] := 317.10938, [2325] := 317.19727, [2326] := 317.37305, [2327] := 317.28516, [2328] := 316.40625, [2329] := 316.49414, [2330] := 316.66992, [2331] := 316.58203, [2332] := 317.02148, [2333] := 316.9336, [2334] := 316.7578, [2335] := 316.8457, [2336] := 320.5371, [2337] := 320.44922, [2338] := 320.27344, [2339] := 320.36133, [2340] := 319.92188,
        [2341] := 320.00977, [2342] := 320.18555, [2343] := 320.09766, [2344] := 319.21875, [2345] := 319.30664, [2346] := 319.48242, [2347] := 319.39453, [2348] := 319.83398, [2349] := 319.7461, [2350] := 319.5703, [2351] := 319.6582, [2352] := 317.8125, [2353] := 317.9004, [2354] := 318.07617, [2355] := 317.98828, [2356] := 318.42773, [2357] := 318.33984, [2358] := 318.16406, [2359] := 318.25195, [2360] := 319.13086, [2361] := 319.04297, [2362] := 318.8672, [2363] := 318.95508, [2364] := 318.51562, [2365] := 318.60352, [2366] := 318.7793, [2367] := 318.6914, [2368] := 326.1621, [2369] := 326.07422, [2370] := 325.89844, [2371] := 325.98633, [2372] := 325.54688, [2373] := 325.63477, [2374] := 325.81055, [2375] := 325.72266, [2376] := 324.84375, [2377] := 324.93164, [2378] := 325.10742, [2379] := 325.01953, [2380] := 325.45898, [2381] := 325.3711, [2382] := 325.1953, [2383] := 325.2832, [2384] := 323.4375, [2385] := 323.5254, [2386] := 323.70117, [2387] := 323.61328, [2388] := 324.05273, [2389] := 323.96484, [2390] := 323.78906, [2391] := 323.87695, [2392] := 324.75586, [2393] := 324.66797, [2394] := 324.4922, [2395] := 324.58008, [2396] := 324.14062, [2397] := 324.22852, [2398] := 324.4043, [2399] := 324.3164, [2400] := 320.625,
        [2401] := 320.7129, [2402] := 320.88867, [2403] := 320.80078, [2404] := 321.24023, [2405] := 321.15234, [2406] := 320.97656, [2407] := 321.06445, [2408] := 321.94336, [2409] := 321.85547, [2410] := 321.6797, [2411] := 321.76758, [2412] := 321.32812, [2413] := 321.41602, [2414] := 321.5918, [2415] := 321.5039, [2416] := 323.3496, [2417] := 323.26172, [2418] := 323.08594, [2419] := 323.17383, [2420] := 322.73438, [2421] := 322.82227, [2422] := 322.99805, [2423] := 322.91016, [2424] := 322.03125, [2425] := 322.11914, [2426] := 322.29492, [2427] := 322.20703, [2428] := 322.64648, [2429] := 322.5586, [2430] := 322.3828, [2431] := 322.4707, [2432] := 337.4121, [2433] := 337.32422, [2434] := 337.14844, [2435] := 337.23633, [2436] := 336.79688, [2437] := 336.88477, [2438] := 337.06055, [2439] := 336.97266, [2440] := 336.09375, [2441] := 336.18164, [2442] := 336.35742, [2443] := 336.26953, [2444] := 336.70898, [2445] := 336.6211, [2446] := 336.4453, [2447] := 336.5332, [2448] := 334.6875, [2449] := 334.7754, [2450] := 334.95117, [2451] := 334.86328, [2452] := 335.30273, [2453] := 335.21484, [2454] := 335.03906, [2455] := 335.12695, [2456] := 336.00586, [2457] := 335.91797, [2458] := 335.7422, [2459] := 335.83008, [2460] := 335.39062,
        [2461] := 335.47852, [2462] := 335.6543, [2463] := 335.5664, [2464] := 331.875, [2465] := 331.9629, [2466] := 332.13867, [2467] := 332.05078, [2468] := 332.49023, [2469] := 332.40234, [2470] := 332.22656, [2471] := 332.31445, [2472] := 333.19336, [2473] := 333.10547, [2474] := 332.9297, [2475] := 333.01758, [2476] := 332.57812, [2477] := 332.66602, [2478] := 332.8418, [2479] := 332.7539, [2480] := 334.5996, [2481] := 334.51172, [2482] := 334.33594, [2483] := 334.42383, [2484] := 333.98438, [2485] := 334.07227, [2486] := 334.24805, [2487] := 334.16016, [2488] := 333.28125, [2489] := 333.36914, [2490] := 333.54492, [2491] := 333.45703, [2492] := 333.89648, [2493] := 333.8086, [2494] := 333.6328, [2495] := 333.7207, [2496] := 326.25, [2497] := 326.3379, [2498] := 326.51367, [2499] := 326.42578, [2500] := 326.86523, [2501] := 326.77734, [2502] := 326.60156, [2503] := 326.68945, [2504] := 327.56836, [2505] := 327.48047, [2506] := 327.3047, [2507] := 327.39258, [2508] := 326.95312, [2509] := 327.04102, [2510] := 327.2168, [2511] := 327.1289, [2512] := 328.9746, [2513] := 328.88672, [2514] := 328.71094, [2515] := 328.79883, [2516] := 328.35938, [2517] := 328.44727, [2518] := 328.62305, [2519] := 328.53516, [2520] := 327.65625,
        [2521] := 327.74414, [2522] := 327.91992, [2523] := 327.83203, [2524] := 328.27148, [2525] := 328.1836, [2526] := 328.0078, [2527] := 328.0957, [2528] := 331.7871, [2529] := 331.69922, [2530] := 331.52344, [2531] := 331.61133, [2532] := 331.17188, [2533] := 331.25977, [2534] := 331.43555, [2535] := 331.34766, [2536] := 330.46875, [2537] := 330.55664, [2538] := 330.73242, [2539] := 330.64453, [2540] := 331.08398, [2541] := 330.9961, [2542] := 330.8203, [2543] := 330.9082, [2544] := 329.0625, [2545] := 329.1504, [2546] := 329.32617, [2547] := 329.23828, [2548] := 329.67773, [2549] := 329.58984, [2550] := 329.41406, [2551] := 329.50195, [2552] := 330.38086, [2553] := 330.29297, [2554] := 330.1172, [2555] := 330.20508, [2556] := 329.76562, [2557] := 329.85352, [2558] := 330.0293, [2559] := 329.9414, [2560] := 270.0, [2561] := 270.0879, [2562] := 270.26367, [2563] := 270.17578, [2564] := 270.61523, [2565] := 270.52734, [2566] := 270.35156, [2567] := 270.43945, [2568] := 271.31836, [2569] := 271.23047, [2570] := 271.0547, [2571] := 271.14258, [2572] := 270.70312, [2573] := 270.79102, [2574] := 270.9668, [2575] := 270.8789, [2576] := 272.7246, [2577] := 272.63672, [2578] := 272.46094, [2579] := 272.54883, [2580] := 272.10938,
        [2581] := 272.19727, [2582] := 272.37305, [2583] := 272.28516, [2584] := 271.40625, [2585] := 271.49414, [2586] := 271.66992, [2587] := 271.58203, [2588] := 272.02148, [2589] := 271.9336, [2590] := 271.7578, [2591] := 271.8457, [2592] := 275.5371, [2593] := 275.44922, [2594] := 275.27344, [2595] := 275.36133, [2596] := 274.92188, [2597] := 275.00977, [2598] := 275.18555, [2599] := 275.09766, [2600] := 274.21875, [2601] := 274.30664, [2602] := 274.48242, [2603] := 274.39453, [2604] := 274.83398, [2605] := 274.7461, [2606] := 274.5703, [2607] := 274.6582, [2608] := 272.8125, [2609] := 272.9004, [2610] := 273.07617, [2611] := 272.98828, [2612] := 273.42773, [2613] := 273.33984, [2614] := 273.16406, [2615] := 273.25195, [2616] := 274.13086, [2617] := 274.04297, [2618] := 273.8672, [2619] := 273.95508, [2620] := 273.51562, [2621] := 273.60352, [2622] := 273.7793, [2623] := 273.6914, [2624] := 281.1621, [2625] := 281.07422, [2626] := 280.89844, [2627] := 280.98633, [2628] := 280.54688, [2629] := 280.63477, [2630] := 280.81055, [2631] := 280.72266, [2632] := 279.84375, [2633] := 279.93164, [2634] := 280.10742, [2635] := 280.01953, [2636] := 280.45898, [2637] := 280.3711, [2638] := 280.1953, [2639] := 280.2832, [2640] := 278.4375,
        [2641] := 278.5254, [2642] := 278.70117, [2643] := 278.61328, [2644] := 279.05273, [2645] := 278.96484, [2646] := 278.78906, [2647] := 278.87695, [2648] := 279.75586, [2649] := 279.66797, [2650] := 279.4922, [2651] := 279.58008, [2652] := 279.14062, [2653] := 279.22852, [2654] := 279.4043, [2655] := 279.3164, [2656] := 275.625, [2657] := 275.7129, [2658] := 275.88867, [2659] := 275.80078, [2660] := 276.24023, [2661] := 276.15234, [2662] := 275.97656, [2663] := 276.06445, [2664] := 276.94336, [2665] := 276.85547, [2666] := 276.6797, [2667] := 276.76758, [2668] := 276.32812, [2669] := 276.41602, [2670] := 276.5918, [2671] := 276.5039, [2672] := 278.3496, [2673] := 278.26172, [2674] := 278.08594, [2675] := 278.17383, [2676] := 277.73438, [2677] := 277.82227, [2678] := 277.99805, [2679] := 277.91016, [2680] := 277.03125, [2681] := 277.11914, [2682] := 277.29492, [2683] := 277.20703, [2684] := 277.64648, [2685] := 277.5586, [2686] := 277.3828, [2687] := 277.4707, [2688] := 292.4121, [2689] := 292.32422, [2690] := 292.14844, [2691] := 292.23633, [2692] := 291.79688, [2693] := 291.88477, [2694] := 292.06055, [2695] := 291.97266, [2696] := 291.09375, [2697] := 291.18164, [2698] := 291.35742, [2699] := 291.26953, [2700] := 291.70898,
        [2701] := 291.6211, [2702] := 291.4453, [2703] := 291.5332, [2704] := 289.6875, [2705] := 289.7754, [2706] := 289.95117, [2707] := 289.86328, [2708] := 290.30273, [2709] := 290.21484, [2710] := 290.03906, [2711] := 290.12695, [2712] := 291.00586, [2713] := 290.91797, [2714] := 290.7422, [2715] := 290.83008, [2716] := 290.39062, [2717] := 290.47852, [2718] := 290.6543, [2719] := 290.5664, [2720] := 286.875, [2721] := 286.9629, [2722] := 287.13867, [2723] := 287.05078, [2724] := 287.49023, [2725] := 287.40234, [2726] := 287.22656, [2727] := 287.31445, [2728] := 288.19336, [2729] := 288.10547, [2730] := 287.9297, [2731] := 288.01758, [2732] := 287.57812, [2733] := 287.66602, [2734] := 287.8418, [2735] := 287.7539, [2736] := 289.5996, [2737] := 289.51172, [2738] := 289.33594, [2739] := 289.42383, [2740] := 288.98438, [2741] := 289.07227, [2742] := 289.24805, [2743] := 289.16016, [2744] := 288.28125, [2745] := 288.36914, [2746] := 288.54492, [2747] := 288.45703, [2748] := 288.89648, [2749] := 288.8086, [2750] := 288.6328, [2751] := 288.7207, [2752] := 281.25, [2753] := 281.3379, [2754] := 281.51367, [2755] := 281.42578, [2756] := 281.86523, [2757] := 281.77734, [2758] := 281.60156, [2759] := 281.68945, [2760] := 282.56836,
        [2761] := 282.48047, [2762] := 282.3047, [2763] := 282.39258, [2764] := 281.95312, [2765] := 282.04102, [2766] := 282.2168, [2767] := 282.1289, [2768] := 283.9746, [2769] := 283.88672, [2770] := 283.71094, [2771] := 283.79883, [2772] := 283.35938, [2773] := 283.44727, [2774] := 283.62305, [2775] := 283.53516, [2776] := 282.65625, [2777] := 282.74414, [2778] := 282.91992, [2779] := 282.83203, [2780] := 283.27148, [2781] := 283.1836, [2782] := 283.0078, [2783] := 283.0957, [2784] := 286.7871, [2785] := 286.69922, [2786] := 286.52344, [2787] := 286.61133, [2788] := 286.17188, [2789] := 286.25977, [2790] := 286.43555, [2791] := 286.34766, [2792] := 285.46875, [2793] := 285.55664, [2794] := 285.73242, [2795] := 285.64453, [2796] := 286.08398, [2797] := 285.9961, [2798] := 285.8203, [2799] := 285.9082, [2800] := 284.0625, [2801] := 284.1504, [2802] := 284.32617, [2803] := 284.23828, [2804] := 284.67773, [2805] := 284.58984, [2806] := 284.41406, [2807] := 284.50195, [2808] := 285.38086, [2809] := 285.29297, [2810] := 285.1172, [2811] := 285.20508, [2812] := 284.76562, [2813] := 284.85352, [2814] := 285.0293, [2815] := 284.9414, [2816] := 314.9121, [2817] := 314.82422, [2818] := 314.64844, [2819] := 314.73633, [2820] := 314.29688,
        [2821] := 314.38477, [2822] := 314.56055, [2823] := 314.47266, [2824] := 313.59375, [2825] := 313.68164, [2826] := 313.85742, [2827] := 313.76953, [2828] := 314.20898, [2829] := 314.1211, [2830] := 313.9453, [2831] := 314.0332, [2832] := 312.1875, [2833] := 312.2754, [2834] := 312.45117, [2835] := 312.36328, [2836] := 312.80273, [2837] := 312.71484, [2838] := 312.53906, [2839] := 312.62695, [2840] := 313.50586, [2841] := 313.41797, [2842] := 313.2422, [2843] := 313.33008, [2844] := 312.89062, [2845] := 312.97852, [2846] := 313.1543, [2847] := 313.0664, [2848] := 309.375, [2849] := 309.4629, [2850] := 309.63867, [2851] := 309.55078, [2852] := 309.99023, [2853] := 309.90234, [2854] := 309.72656, [2855] := 309.81445, [2856] := 310.69336, [2857] := 310.60547, [2858] := 310.4297, [2859] := 310.51758, [2860] := 310.07812, [2861] := 310.16602, [2862] := 310.3418, [2863] := 310.2539, [2864] := 312.0996, [2865] := 312.01172, [2866] := 311.83594, [2867] := 311.92383, [2868] := 311.48438, [2869] := 311.57227, [2870] := 311.74805, [2871] := 311.66016, [2872] := 310.78125, [2873] := 310.86914, [2874] := 311.04492, [2875] := 310.95703, [2876] := 311.39648, [2877] := 311.3086, [2878] := 311.1328, [2879] := 311.2207, [2880] := 303.75,
        [2881] := 303.8379, [2882] := 304.01367, [2883] := 303.92578, [2884] := 304.36523, [2885] := 304.27734, [2886] := 304.10156, [2887] := 304.18945, [2888] := 305.06836, [2889] := 304.98047, [2890] := 304.8047, [2891] := 304.89258, [2892] := 304.45312, [2893] := 304.54102, [2894] := 304.7168, [2895] := 304.6289, [2896] := 306.4746, [2897] := 306.38672, [2898] := 306.21094, [2899] := 306.29883, [2900] := 305.85938, [2901] := 305.94727, [2902] := 306.12305, [2903] := 306.03516, [2904] := 305.15625, [2905] := 305.24414, [2906] := 305.41992, [2907] := 305.33203, [2908] := 305.77148, [2909] := 305.6836, [2910] := 305.5078, [2911] := 305.5957, [2912] := 309.2871, [2913] := 309.19922, [2914] := 309.02344, [2915] := 309.11133, [2916] := 308.67188, [2917] := 308.75977, [2918] := 308.93555, [2919] := 308.84766, [2920] := 307.96875, [2921] := 308.05664, [2922] := 308.23242, [2923] := 308.14453, [2924] := 308.58398, [2925] := 308.4961, [2926] := 308.3203, [2927] := 308.4082, [2928] := 306.5625, [2929] := 306.6504, [2930] := 306.82617, [2931] := 306.73828, [2932] := 307.17773, [2933] := 307.08984, [2934] := 306.91406, [2935] := 307.00195, [2936] := 307.88086, [2937] := 307.79297, [2938] := 307.6172, [2939] := 307.70508, [2940] := 307.26562,
        [2941] := 307.35352, [2942] := 307.5293, [2943] := 307.4414, [2944] := 292.5, [2945] := 292.5879, [2946] := 292.76367, [2947] := 292.67578, [2948] := 293.11523, [2949] := 293.02734, [2950] := 292.85156, [2951] := 292.93945, [2952] := 293.81836, [2953] := 293.73047, [2954] := 293.5547, [2955] := 293.64258, [2956] := 293.20312, [2957] := 293.29102, [2958] := 293.4668, [2959] := 293.3789, [2960] := 295.2246, [2961] := 295.13672, [2962] := 294.96094, [2963] := 295.04883, [2964] := 294.60938, [2965] := 294.69727, [2966] := 294.87305, [2967] := 294.78516, [2968] := 293.90625, [2969] := 293.99414, [2970] := 294.16992, [2971] := 294.08203, [2972] := 294.52148, [2973] := 294.4336, [2974] := 294.2578, [2975] := 294.3457, [2976] := 298.0371, [2977] := 297.94922, [2978] := 297.77344, [2979] := 297.86133, [2980] := 297.42188, [2981] := 297.50977, [2982] := 297.68555, [2983] := 297.59766, [2984] := 296.71875, [2985] := 296.80664, [2986] := 296.98242, [2987] := 296.89453, [2988] := 297.33398, [2989] := 297.2461, [2990] := 297.0703, [2991] := 297.1582, [2992] := 295.3125, [2993] := 295.4004, [2994] := 295.57617, [2995] := 295.48828, [2996] := 295.92773, [2997] := 295.83984, [2998] := 295.66406, [2999] := 295.75195, [3000] := 296.63086,
        [3001] := 296.54297, [3002] := 296.3672, [3003] := 296.45508, [3004] := 296.01562, [3005] := 296.10352, [3006] := 296.2793, [3007] := 296.1914, [3008] := 303.6621, [3009] := 303.57422, [3010] := 303.39844, [3011] := 303.48633, [3012] := 303.04688, [3013] := 303.13477, [3014] := 303.31055, [3015] := 303.22266, [3016] := 302.34375, [3017] := 302.43164, [3018] := 302.60742, [3019] := 302.51953, [3020] := 302.95898, [3021] := 302.8711, [3022] := 302.6953, [3023] := 302.7832, [3024] := 300.9375, [3025] := 301.0254, [3026] := 301.20117, [3027] := 301.11328, [3028] := 301.55273, [3029] := 301.46484, [3030] := 301.28906, [3031] := 301.37695, [3032] := 302.25586, [3033] := 302.16797, [3034] := 301.9922, [3035] := 302.08008, [3036] := 301.64062, [3037] := 301.72852, [3038] := 301.9043, [3039] := 301.8164, [3040] := 298.125, [3041] := 298.2129, [3042] := 298.38867, [3043] := 298.30078, [3044] := 298.74023, [3045] := 298.65234, [3046] := 298.47656, [3047] := 298.56445, [3048] := 299.44336, [3049] := 299.35547, [3050] := 299.1797, [3051] := 299.26758, [3052] := 298.82812, [3053] := 298.91602, [3054] := 299.0918, [3055] := 299.0039, [3056] := 300.8496, [3057] := 300.76172, [3058] := 300.58594, [3059] := 300.67383, [3060] := 300.23438,
        [3061] := 300.32227, [3062] := 300.49805, [3063] := 300.41016, [3064] := 299.53125, [3065] := 299.61914, [3066] := 299.79492, [3067] := 299.70703, [3068] := 300.14648, [3069] := 300.0586, [3070] := 299.8828, [3071] := 299.9707, [3072] := 180.0, [3073] := 180.08789, [3074] := 180.26367, [3075] := 180.17578, [3076] := 180.61523, [3077] := 180.52734, [3078] := 180.35156, [3079] := 180.43945, [3080] := 181.31836, [3081] := 181.23047, [3082] := 181.05469, [3083] := 181.14258, [3084] := 180.70312, [3085] := 180.79102, [3086] := 180.9668, [3087] := 180.8789, [3088] := 182.72461, [3089] := 182.63672, [3090] := 182.46094, [3091] := 182.54883, [3092] := 182.10938, [3093] := 182.19727, [3094] := 182.37305, [3095] := 182.28516, [3096] := 181.40625, [3097] := 181.49414, [3098] := 181.66992, [3099] := 181.58203, [3100] := 182.02148, [3101] := 181.9336, [3102] := 181.75781, [3103] := 181.8457, [3104] := 185.53711, [3105] := 185.44922, [3106] := 185.27344, [3107] := 185.36133, [3108] := 184.92188, [3109] := 185.00977, [3110] := 185.18555, [3111] := 185.09766, [3112] := 184.21875, [3113] := 184.30664, [3114] := 184.48242, [3115] := 184.39453, [3116] := 184.83398, [3117] := 184.7461, [3118] := 184.57031, [3119] := 184.6582, [3120] := 182.8125,
        [3121] := 182.90039, [3122] := 183.07617, [3123] := 182.98828, [3124] := 183.42773, [3125] := 183.33984, [3126] := 183.16406, [3127] := 183.25195, [3128] := 184.13086, [3129] := 184.04297, [3130] := 183.86719, [3131] := 183.95508, [3132] := 183.51562, [3133] := 183.60352, [3134] := 183.7793, [3135] := 183.6914, [3136] := 191.16211, [3137] := 191.07422, [3138] := 190.89844, [3139] := 190.98633, [3140] := 190.54688, [3141] := 190.63477, [3142] := 190.81055, [3143] := 190.72266, [3144] := 189.84375, [3145] := 189.93164, [3146] := 190.10742, [3147] := 190.01953, [3148] := 190.45898, [3149] := 190.3711, [3150] := 190.19531, [3151] := 190.2832, [3152] := 188.4375, [3153] := 188.52539, [3154] := 188.70117, [3155] := 188.61328, [3156] := 189.05273, [3157] := 188.96484, [3158] := 188.78906, [3159] := 188.87695, [3160] := 189.75586, [3161] := 189.66797, [3162] := 189.49219, [3163] := 189.58008, [3164] := 189.14062, [3165] := 189.22852, [3166] := 189.4043, [3167] := 189.3164, [3168] := 185.625, [3169] := 185.71289, [3170] := 185.88867, [3171] := 185.80078, [3172] := 186.24023, [3173] := 186.15234, [3174] := 185.97656, [3175] := 186.06445, [3176] := 186.94336, [3177] := 186.85547, [3178] := 186.67969, [3179] := 186.76758, [3180] := 186.32812,
        [3181] := 186.41602, [3182] := 186.5918, [3183] := 186.5039, [3184] := 188.34961, [3185] := 188.26172, [3186] := 188.08594, [3187] := 188.17383, [3188] := 187.73438, [3189] := 187.82227, [3190] := 187.99805, [3191] := 187.91016, [3192] := 187.03125, [3193] := 187.11914, [3194] := 187.29492, [3195] := 187.20703, [3196] := 187.64648, [3197] := 187.5586, [3198] := 187.38281, [3199] := 187.4707, [3200] := 202.41211, [3201] := 202.32422, [3202] := 202.14844, [3203] := 202.23633, [3204] := 201.79688, [3205] := 201.88477, [3206] := 202.06055, [3207] := 201.97266, [3208] := 201.09375, [3209] := 201.18164, [3210] := 201.35742, [3211] := 201.26953, [3212] := 201.70898, [3213] := 201.6211, [3214] := 201.44531, [3215] := 201.5332, [3216] := 199.6875, [3217] := 199.77539, [3218] := 199.95117, [3219] := 199.86328, [3220] := 200.30273, [3221] := 200.21484, [3222] := 200.03906, [3223] := 200.12695, [3224] := 201.00586, [3225] := 200.91797, [3226] := 200.74219, [3227] := 200.83008, [3228] := 200.39062, [3229] := 200.47852, [3230] := 200.6543, [3231] := 200.5664, [3232] := 196.875, [3233] := 196.96289, [3234] := 197.13867, [3235] := 197.05078, [3236] := 197.49023, [3237] := 197.40234, [3238] := 197.22656, [3239] := 197.31445, [3240] := 198.19336,
        [3241] := 198.10547, [3242] := 197.92969, [3243] := 198.01758, [3244] := 197.57812, [3245] := 197.66602, [3246] := 197.8418, [3247] := 197.7539, [3248] := 199.59961, [3249] := 199.51172, [3250] := 199.33594, [3251] := 199.42383, [3252] := 198.98438, [3253] := 199.07227, [3254] := 199.24805, [3255] := 199.16016, [3256] := 198.28125, [3257] := 198.36914, [3258] := 198.54492, [3259] := 198.45703, [3260] := 198.89648, [3261] := 198.8086, [3262] := 198.63281, [3263] := 198.7207, [3264] := 191.25, [3265] := 191.33789, [3266] := 191.51367, [3267] := 191.42578, [3268] := 191.86523, [3269] := 191.77734, [3270] := 191.60156, [3271] := 191.68945, [3272] := 192.56836, [3273] := 192.48047, [3274] := 192.30469, [3275] := 192.39258, [3276] := 191.95312, [3277] := 192.04102, [3278] := 192.2168, [3279] := 192.1289, [3280] := 193.97461, [3281] := 193.88672, [3282] := 193.71094, [3283] := 193.79883, [3284] := 193.35938, [3285] := 193.44727, [3286] := 193.62305, [3287] := 193.53516, [3288] := 192.65625, [3289] := 192.74414, [3290] := 192.91992, [3291] := 192.83203, [3292] := 193.27148, [3293] := 193.1836, [3294] := 193.00781, [3295] := 193.0957, [3296] := 196.78711, [3297] := 196.69922, [3298] := 196.52344, [3299] := 196.61133, [3300] := 196.17188,
        [3301] := 196.25977, [3302] := 196.43555, [3303] := 196.34766, [3304] := 195.46875, [3305] := 195.55664, [3306] := 195.73242, [3307] := 195.64453, [3308] := 196.08398, [3309] := 195.9961, [3310] := 195.82031, [3311] := 195.9082, [3312] := 194.0625, [3313] := 194.15039, [3314] := 194.32617, [3315] := 194.23828, [3316] := 194.67773, [3317] := 194.58984, [3318] := 194.41406, [3319] := 194.50195, [3320] := 195.38086, [3321] := 195.29297, [3322] := 195.11719, [3323] := 195.20508, [3324] := 194.76562, [3325] := 194.85352, [3326] := 195.0293, [3327] := 194.9414, [3328] := 224.91211, [3329] := 224.82422, [3330] := 224.64844, [3331] := 224.73633, [3332] := 224.29688, [3333] := 224.38477, [3334] := 224.56055, [3335] := 224.47266, [3336] := 223.59375, [3337] := 223.68164, [3338] := 223.85742, [3339] := 223.76953, [3340] := 224.20898, [3341] := 224.1211, [3342] := 223.94531, [3343] := 224.0332, [3344] := 222.1875, [3345] := 222.27539, [3346] := 222.45117, [3347] := 222.36328, [3348] := 222.80273, [3349] := 222.71484, [3350] := 222.53906, [3351] := 222.62695, [3352] := 223.50586, [3353] := 223.41797, [3354] := 223.24219, [3355] := 223.33008, [3356] := 222.89062, [3357] := 222.97852, [3358] := 223.1543, [3359] := 223.0664, [3360] := 219.375,
        [3361] := 219.46289, [3362] := 219.63867, [3363] := 219.55078, [3364] := 219.99023, [3365] := 219.90234, [3366] := 219.72656, [3367] := 219.81445, [3368] := 220.69336, [3369] := 220.60547, [3370] := 220.42969, [3371] := 220.51758, [3372] := 220.07812, [3373] := 220.16602, [3374] := 220.3418, [3375] := 220.2539, [3376] := 222.09961, [3377] := 222.01172, [3378] := 221.83594, [3379] := 221.92383, [3380] := 221.48438, [3381] := 221.57227, [3382] := 221.74805, [3383] := 221.66016, [3384] := 220.78125, [3385] := 220.86914, [3386] := 221.04492, [3387] := 220.95703, [3388] := 221.39648, [3389] := 221.3086, [3390] := 221.13281, [3391] := 221.2207, [3392] := 213.75, [3393] := 213.83789, [3394] := 214.01367, [3395] := 213.92578, [3396] := 214.36523, [3397] := 214.27734, [3398] := 214.10156, [3399] := 214.18945, [3400] := 215.06836, [3401] := 214.98047, [3402] := 214.80469, [3403] := 214.89258, [3404] := 214.45312, [3405] := 214.54102, [3406] := 214.7168, [3407] := 214.6289, [3408] := 216.47461, [3409] := 216.38672, [3410] := 216.21094, [3411] := 216.29883, [3412] := 215.85938, [3413] := 215.94727, [3414] := 216.12305, [3415] := 216.03516, [3416] := 215.15625, [3417] := 215.24414, [3418] := 215.41992, [3419] := 215.33203, [3420] := 215.77148,
        [3421] := 215.6836, [3422] := 215.50781, [3423] := 215.5957, [3424] := 219.28711, [3425] := 219.19922, [3426] := 219.02344, [3427] := 219.11133, [3428] := 218.67188, [3429] := 218.75977, [3430] := 218.93555, [3431] := 218.84766, [3432] := 217.96875, [3433] := 218.05664, [3434] := 218.23242, [3435] := 218.14453, [3436] := 218.58398, [3437] := 218.4961, [3438] := 218.32031, [3439] := 218.4082, [3440] := 216.5625, [3441] := 216.65039, [3442] := 216.82617, [3443] := 216.73828, [3444] := 217.17773, [3445] := 217.08984, [3446] := 216.91406, [3447] := 217.00195, [3448] := 217.88086, [3449] := 217.79297, [3450] := 217.61719, [3451] := 217.70508, [3452] := 217.26562, [3453] := 217.35352, [3454] := 217.5293, [3455] := 217.4414, [3456] := 202.5, [3457] := 202.58789, [3458] := 202.76367, [3459] := 202.67578, [3460] := 203.11523, [3461] := 203.02734, [3462] := 202.85156, [3463] := 202.93945, [3464] := 203.81836, [3465] := 203.73047, [3466] := 203.55469, [3467] := 203.64258, [3468] := 203.20312, [3469] := 203.29102, [3470] := 203.4668, [3471] := 203.3789, [3472] := 205.22461, [3473] := 205.13672, [3474] := 204.96094, [3475] := 205.04883, [3476] := 204.60938, [3477] := 204.69727, [3478] := 204.87305, [3479] := 204.78516, [3480] := 203.90625,
        [3481] := 203.99414, [3482] := 204.16992, [3483] := 204.08203, [3484] := 204.52148, [3485] := 204.4336, [3486] := 204.25781, [3487] := 204.3457, [3488] := 208.03711, [3489] := 207.94922, [3490] := 207.77344, [3491] := 207.86133, [3492] := 207.42188, [3493] := 207.50977, [3494] := 207.68555, [3495] := 207.59766, [3496] := 206.71875, [3497] := 206.80664, [3498] := 206.98242, [3499] := 206.89453, [3500] := 207.33398, [3501] := 207.2461, [3502] := 207.07031, [3503] := 207.1582, [3504] := 205.3125, [3505] := 205.40039, [3506] := 205.57617, [3507] := 205.48828, [3508] := 205.92773, [3509] := 205.83984, [3510] := 205.66406, [3511] := 205.75195, [3512] := 206.63086, [3513] := 206.54297, [3514] := 206.36719, [3515] := 206.45508, [3516] := 206.01562, [3517] := 206.10352, [3518] := 206.2793, [3519] := 206.1914, [3520] := 213.66211, [3521] := 213.57422, [3522] := 213.39844, [3523] := 213.48633, [3524] := 213.04688, [3525] := 213.13477, [3526] := 213.31055, [3527] := 213.22266, [3528] := 212.34375, [3529] := 212.43164, [3530] := 212.60742, [3531] := 212.51953, [3532] := 212.95898, [3533] := 212.8711, [3534] := 212.69531, [3535] := 212.7832, [3536] := 210.9375, [3537] := 211.02539, [3538] := 211.20117, [3539] := 211.11328, [3540] := 211.55273,
        [3541] := 211.46484, [3542] := 211.28906, [3543] := 211.37695, [3544] := 212.25586, [3545] := 212.16797, [3546] := 211.99219, [3547] := 212.08008, [3548] := 211.64062, [3549] := 211.72852, [3550] := 211.9043, [3551] := 211.8164, [3552] := 208.125, [3553] := 208.21289, [3554] := 208.38867, [3555] := 208.30078, [3556] := 208.74023, [3557] := 208.65234, [3558] := 208.47656, [3559] := 208.56445, [3560] := 209.44336, [3561] := 209.35547, [3562] := 209.17969, [3563] := 209.26758, [3564] := 208.82812, [3565] := 208.91602, [3566] := 209.0918, [3567] := 209.0039, [3568] := 210.84961, [3569] := 210.76172, [3570] := 210.58594, [3571] := 210.67383, [3572] := 210.23438, [3573] := 210.32227, [3574] := 210.49805, [3575] := 210.41016, [3576] := 209.53125, [3577] := 209.61914, [3578] := 209.79492, [3579] := 209.70703, [3580] := 210.14648, [3581] := 210.0586, [3582] := 209.88281, [3583] := 209.9707, [3584] := 269.9121, [3585] := 269.82422, [3586] := 269.64844, [3587] := 269.73633, [3588] := 269.29688, [3589] := 269.38477, [3590] := 269.56055, [3591] := 269.47266, [3592] := 268.59375, [3593] := 268.68164, [3594] := 268.85742, [3595] := 268.76953, [3596] := 269.20898, [3597] := 269.1211, [3598] := 268.9453, [3599] := 269.0332, [3600] := 267.1875,
